FUNCTION_BLOCK FB_MachineControl EXTENDS FB_UniversalMachine IMPLEMENTS I_MachineControl
VAR PERSISTENT
	sLastLoadedRecipe						: STRING;
	sLastProductOrder						: STRING;
	(* Parameter have to adjust for Sorting Station *)
	lrSortGoodDistance			: LREAL := -24.0;	(* Distance between cam7 to sort station *)
	lrSortDirtDistance			: LREAL := -55.0;	(* Distance between cam7 to sort station *)
	lrSortDentDistance			: LREAL := -55.0;	(* Distance between cam7 to sort station *)
	lrSortRejectDistance		: LREAL := -60.0;	(* Distance between cam7 to sort station *)
	tSortValveGoodTime			: TIME := T#1000MS;		(* During time to shoot sample *)
	tSortValveDirtTime			: TIME := T#2000MS;		(* During time to shoot sample *)
	tSortValveDentTime			: TIME := T#1000MS;		(* During time to shoot sample *)
	tSortValveRejectTime		: TIME := T#1000MS;		(* During time to shoot sample *)
	
	rBowlFeederSetpoint 		: REAL := 60.0;
END_VAR
VAR	
	(* Process data *)
	//{attribute 'OPC.UA.DA' := '1	'}
	stBatchPerformance		: ST_BatchPerformacne; 	(* Data about performance about current proccesed batch *)
	//{attribute 'OPC.UA.DA' := '1	'}                                                          		
	stBatchData				: ST_BatchData;			(* Data about batch that is going to be processed*)

	(*--- Module Interface ---*)
	fbRobot 					: FB_Robot;
	fbRTCVision 				: FB_RTCVision;
	fbBowlFeeder				: FB_BowlFeeder;
	fbRotaryTable				: FB_AxisServo;
	
	(* Utilities *)
	fbPlcUps					: FB_UpsCx51xx;	
	
	(* IO PLC connect *)
	diProductPresenceBowl		: FB_DigitalInput;	(* *)
	diProductPresenceRobot		: FB_DigitalInput;	(* *)	
	
	poDoorLock					: FB_DigitalOutput;			(* Requests all machine lock's to close *)
	poResetButtonLight			: FB_DigitalOutput;			(* Physical reset button attached to door's of electrical cabinet *)
	
	doBlowBowlFeeder			: FB_DigitalOutput;
	doBlowGood					: FB_DigitalOutput;
	doBlowReject				: FB_DigitalOutput;
	doBlowDentContamination		: FB_DigitalOutput;
	doBlowDirtScratch			: FB_DigitalOutput;
	
	doTriggerCam1				: FB_DoubleTrigger;
	doTriggerCam2				: FB_DoubleTrigger;
	doTriggerCam3				: FB_DoubleTrigger;
	doTriggerCam4				: FB_DoubleTrigger;
	doTriggerCam5				: FB_DoubleTrigger;
	doTriggerCam6				: FB_DoubleTrigger;
	doTriggerCam7				: FB_DoubleTrigger;
	
	
	
	(* Auxilary *)
	tonDelay					: TON;				(* Provides any delay into the machine when switching something On/Off *)
	//tonTestDelay	: TON;	(* Delay which allows to see any page changes during tests *)	
	
	(* Parameter *)
	lrHOME_POSTION				: LREAL := 0.0;		(* Homming position *)
	stRotaryTableHomingOptions	: ST_HomingOptions;
	
	(* #ManualToAuto *)             	                                                            		
	//bManualToAutoRotate					: BOOL;																            	
	bStop								: BOOL;	
		
	// =============== State machine ============================================================
	eMachineStateUninitialized						: E_MachineCtrlStateUninitialized;
	eMachineStateInit								: E_MachineCtrlStateInit;
	eMachineStateAuto								: E_MachineCtrlStateAuto;
	eMachineStateAutoAOI							: E_MachineCtrlStateAutoAOI;
	eMachineStateAbort								: E_MachineCtrlStateAbort;
	eMachineStateManualToAuto						: E_MachineCtrlStateManualToAuto;
	
	(* HMI control *)
	btnStartBowl : BOOL;
	btnStopBowl : BOOL;
	
END_VAR

IF bFirstCycle THEN
	(* - bFirstCycle bit reset by parent *)
	(* --- Assign initial parameters for machine objects ---*)
	(* Assign UPS parameters *)
	fbPlcUps.MR_FirstCycle( 	sName 		:= 'PLC UPS',
								sNetID 		:= '',
								iPlcPort 	:= 851,
								tTimeout 	:= DEFAULT_ADS_TIMEOUT);
								
	(* Assign robots *)
	fbRobot.MR_FirstCycle(	sName				:= 'RH-3CRH4018-D-S15',
							iInitialOverride 	:= 3,					//low for testing
							sPLC_NET_ID 		:= '5.127.48.56.2.1',
							iCR800_1_ADDRESS 	:= 1020);
	
	(* Assign rotary table *)
	fbRotaryTable.MR_FirstCycle(	sName				:= sROTARY_TABLE_NAME,
									sMeasurementUnits	:= sROTARY_TABLE_MEASUREMENT_UNIT,
									bModulo				:= FALSE);
									
	fbRotaryTable.Override 			:= 100.0;
	fbRotaryTable.Velocity 			:= 100.0;	//400,325
	fbRotaryTable.Acceleration 		:= 1500.0; //1500,80|600
	fbRotaryTable.Deceleration 		:= 1500.0; //1500,800|600
	fbRotaryTable.Jerk 				:= 6000.0;//6000.0; //15000,8000|

	fbRotaryTable.JogPosition 		:= 0.0;
	fbRotaryTable.JogVelocity 		:= 300.0;
	fbRotaryTable.JogAcceleration 	:= 800.0;
	fbRotaryTable.JogDeceleration 	:= 800.0;
	fbRotaryTable.JogJerk 			:= 800.0;
	fbRotaryTable.StopDeceleration	:= 800.0;
	fbRotaryTable.StopJerk 			:= 8000.0;
	
	stRotaryTableHomingOptions.SearchDirection := Tc2_MC2.MC_Direction.MC_Negative_Direction;
	stRotaryTableHomingOptions.SearchVelocity 	:= 12.0;
	stRotaryTableHomingOptions.SyncDirection 	:= Tc2_MC2.MC_Direction.MC_Positive_Direction;
	stRotaryTableHomingOptions.SyncVelocity	:= 10.0;
	
	fbRotaryTable.HomingMode		:= MC_HomingMode.MC_DefaultHoming;
	fbRotaryTable.HomingOptions 	:= stRotaryTableHomingOptions;

	(* Assign bowl feeder *)
	fbBowlFeeder.MR_FirstCycle(sName := 'Bowl Feeder');
	fbBowlFeeder.Setpoint := 60.0;
	
	(* Assign RTC Vision system *)
	fbRTCVision.MR_FirstCycle(	sCameraName 	:= 'RTC Vision System',
								sClientHost		:= '10.20.254.8',
								sClientAmsNetID := '',
								iClientPort 	:= 23,
								tTimeout 		:= T#15S);
	
	(* Digital I/O *)
	diProductPresenceBowl.MR_FirstCycle(	sName := 'Product presence on bowl at pick point',
											sModuleType := '',
											sPortID := '');
											
	diProductPresenceRobot.MR_FirstCycle(	sName := 'Product presence at robot nozzle',
											sModuleType := '',
											sPortID := '');
									
	poDoorLock.MR_FirstCycle(		sName := 'Door lock station 1',
		                         sModuleType := '',
                                 sPortID := '');
								 
	poResetButtonLight.MR_FirstCycle(	sName := 'Reset Button light station 1',
										sModuleType := '',
										sPortID := '');

END_IF

(* Execute parent implementation *)
SUPER^();

(* --- Cyclic run ---*)
(* Cyclic run robots *)
fbRobot();
(* Cyclic run RTC vision *)
fbRTCVision();
(* Cyclic run bowl feeder *)
fbBowlFeeder();
(* Cyclic run rotary table *)
fbRotaryTable();
(* Utilities *)
fbPlcUps();

PROPERTY BowlFeeder : REFERENCE TO FB_BowlFeeder
GET
BowlFeeder REF= fbBowlFeeder;
END_GET
END_PROPERTY

METHOD PROTECTED GoldenSample : BOOL
VAR_INPUT
END_VAR
;
END_METHOD

METHOD PROTECTED M_AutoProcessing
VAR_INST
	(* Equipment module sequences *)
	BowlFeederProcess : UINT;
	RobotProcess : UINT;
	
	RotaryTableProcess : UINT;
	TableRegister		: UINT;
	
	(* Parameters *)
	bIsRobotAtRotaryTable : BOOL;
	OneStep : LREAL := 10.00;
END_VAR
/// ======================= Bowl feeder process ======================= {{{
CASE BowlFeederProcess OF
	0:
		IF fbBowlFeeder.MR_Start() THEN
			BowlFeederProcess := 10;
		END_IF
		
	10:
		;
		
END_CASE
///}}}
/// ======================= Robot process ======================= {{{
CASE RobotProcess OF
	0://IDLE go bowl
		fbRobot.MR_GoBowl();
		IF NOT fbRobot.Busy THEN
			RobotProcess := 5;
		END_IF
		
	5://Goto input
		IF diProductPresenceBowl.In THEN (* waiting product *)
			fbRobot.MR_GoInputProduct();
			IF NOT fbRobot.Busy THEN
				RobotProcess := 6;
			END_IF
		END_IF
	
	6://robot pick
		fbRobot.MR_Pick();
		IF NOT fbRobot.Busy THEN
			RobotProcess := 10;
		END_IF 
		
	10://go to station 1
		fbRobot.MR_GoStation1();
		IF NOT fbRobot.Busy THEN
			RobotProcess := 20;
		END_IF
	20:
		fbRTCVision.M_CommandStation1(DelayTimeForSecondTrigger := T#1MS);
		IF NOT fbRTCVision.Busy THEN
			RobotProcess := 30;
		END_IF
	30:
		fbRobot.MR_GoStation2();
		IF NOT fbRobot.Busy THEN
			RobotProcess := 40;
		END_IF
	40:
		fbRTCVision.M_CommandStation2(DelayTimeForSecondTrigger := T#34MS);
		IF NOT fbRTCVision.Busy THEN
			RobotProcess := 50;
		END_IF
	50:
		fbrobot.MR_GoRotaryTable();
		IF NOT fbrobot.Busy THEN
			RobotProcess:= 60;//waiting drop product
		END_IF
	
END_CASE

IF RobotProcess = 60 THEN
	bIsRobotAtRotaryTable := TRUE;
ELSE
	bIsRobotAtRotaryTable := FALSE;
END_IF

///}}}
///(*======================= Rotary Table process =======================*){{{
(* Product placed and reset robot sequence *)
CASE TableRegister OF
	0://take product from robot
		IF fbRotaryTable.Halted AND bIsRobotAtRotaryTable THEN
			fbrobot.MR_Place();
			IF NOT fbrobot.Busy THEN
				TableRegister := 10;
			END_IF
		END_IF
	10://buffer calc and add process
		IF Buffer_RotaryTable.Add2Data(in1 := fbRotaryTable.ActualPosition + OneStep, in2 := fbRotaryTable.ActualPosition + 2*OneStep) THEN
			IF Buffer_Station3.Add1Data(in := fbRotaryTable.ActualPosition + OneStep) THEN
				IF Buffer_Station4.Add1Data(in := fbRotaryTable.ActualPosition + 2*OneStep) THEN
					TableRegister := 20;

				END_IF				
			END_IF
		END_IF
END_CASE


(* Table sequences *)
CASE RotaryTableProcess OF
	0://Idle
		IF Buffer_RotaryTable.Count > 0 THEN
			RotaryTableProcess := 10;
		END_IF
	10:
		fbRotaryTable.MR_MoveRelative(lrRelativeDistance := Buffer_RotaryTable.GetValue);
		IF NOT fbRotaryTable.Busy THEN
//			iRTCVision.M_CommandStation1(); // change to station 3
//			IF NOT iRTCVision.Busy THEN
//				;
//			END_IF
			;
		END_IF
END_CASE
///}}}
END_METHOD

METHOD MR_Start : BOOL
(* 
Button START on the HMI
*)
fbMsgAutoStarted.Send(0);

IF eMachineStateAuto = MACHINE_STATE_AUTO_IDLE THEN
	eMachineState := MACHINE_STATE_AUTO;
	eMachineStateAuto := MACHINE_STATE_AUTO_RUNNING;
	bStop := FALSE;
	
END_IF

MR_Start := TRUE;
END_METHOD

METHOD MR_Stop : BOOL
VAR_INPUT
END_VAR
bRunning := FALSE;

IF eMachineStateAuto = MACHINE_STATE_AUTO_RUNNING THEN
	eMachineStateAuto := MACHINE_STATE_AUTO_IDLE;
	
END_IF
END_METHOD

METHOD PROTECTED MS_Aborting
(* 
Add here code to abort all machine objects's e.g robots, axes, cylinders. 
At the end add "eMachineState := MACHINE_STATE_UNINITIALIZED;" to finish aborting.
*)
CASE eMachineStateAbort OF
	MACHINE_STATE_ABORTING_TABLE:
		fbRotaryTable.MR_Abort();
		IF NOT fbRotaryTable.Active THEN
			eMachineState := MACHINE_STATE_UNINITIALIZED;
		eMachineStateUninitialized := MACHINE_STATE_UNINITIALIZED_DONE;
		END_IF
		
	MACHINE_STATE_ABORTING_ROBOT_CYCLE_STOP:
		IF fbRobot.ref_CR800.ErrorOccuring THEN			
			eMachineStateAbort := MACHINE_STATE_ABORTING_TABLE;
			eMachineState := MACHINE_STATE_UNINITIALIZED;
			eMachineStateUninitialized := MACHINE_STATE_UNINITIALIZED_DONE;
		ELSE
			fbRobot.ref_CR800.MR_CycleStop();
			IF NOT fbRobot.ref_CR800.Busy THEN
				eMachineStateAbort := MACHINE_STATE_ABORTING_TABLE;
				eMachineState := MACHINE_STATE_UNINITIALIZED;
				eMachineStateUninitialized := MACHINE_STATE_UNINITIALIZED_DONE;
			END_IF
		END_IF

END_CASE
END_METHOD

METHOD PROTECTED MS_Auto
VAR_INST
	bSetSP:BOOL;
	rSp:REAL;
END_VAR
CASE eMachineStateAuto OF
	MACHINE_STATE_AUTO_IDLE:
		bRunning := FALSE;
		
	MACHINE_STATE_AUTO_RUNNING:
		bRunning := TRUE;
		//Test();
		Production_fixing();
		//Robot_Process();
		//TableProcess();
		//tableRefer();
		//robotcamtest();
		//Robot_Process();
		
END_CASE

(*========== HMI control =============*)
(* Bowl feeder *)
IF btnStartBowl THEN
	fbBowlFeeder.MR_Start();
	doBlowBowlFeeder.Out := TRUE;
END_IF

IF btnStopBowl THEN
	fbBowlFeeder.MR_Stop();
	doBlowBowlFeeder.Out := FALSE;
END_IF

fbBowlFeeder.Setpoint := rBowlFeederSetpoint;
END_METHOD

METHOD PROTECTED MS_AutoToManual
VAR_INPUT
END_VAR
(* 
Add here code to switch machine into manual mode. 
At the end add "eMachineState := MACHINE_STATE_MANUAL;" to finish switching.
*)
(* Switching mode to manual simulation - DELETE *)
//tonTestDelay(IN := TRUE, PT:= T#500MS);
//bRunning := FALSE;
//IF tonTestDelay.Q THEN
//	tonTestDelay(IN := FALSE);
//	eMachineState := MACHINE_STATE_MANUAL;
//END_IF

bRunning := FALSE;
eMachineState := MACHINE_STATE_MANUAL;
END_METHOD

METHOD PROTECTED MS_Emergency
VAR_INPUT
END_VAR
END_METHOD

METHOD PROTECTED MS_Initializing
VAR_INST
	uBowlFeederInitState : UINT;
	uTableInitState : UINT;
	uVisionInitState : UINT;
	
END_VAR
(* 
Add here code to initialize all machine objects's e.g robots, axes, cylinders. 
At the end add "eMachineState := MACHINE_STATE_READY_INITIALIZED;" to finish initialization.
*)
CASE eMachineStateInit OF
	MACHINE_STATE_INITIALIZING_MACHINE_LOGGER:
		fbMachineLogger.MR_Init();
		IF NOT fbMachineLogger.Busy THEN
			eMachineStateInit := MACHINE_STATE_INITIALIZING_ROBOT_CONTROLERS_RESET;
		END_IF
(*	
	MACHINE_STATE_INITIALIZING_RECIPES_MANAGER:
		IF stShell.stPlatform.ref_fbRecipesManager.Active THEN
			eMachineStateInit := MACHINE_STATE_INITIALIZING_CLEAR_ALL_ERRORS;
		END_IF
		
	MACHINE_STATE_INITIALIZING_CLEAR_ALL_ERRORS:
		stShell.stPlatform.ref_fbAlarmControler.MR_ClearAll(TRUE);
		IF NOT stShell.stPlatform.ref_fbAlarmControler.Busy THEN
			//eMachineStateInit := MACHINE_STATE_INITIALIZING_MES_COMMAND_LOGGER;
			eMachineStateInit := MACHINE_STATE_INITIALIZING_SAFETY_INITIALIZATION;
		END_IF
	
	MACHINE_STATE_INITIALIZING_SAFETY_INITIALIZATION:
		stShell.stPlatform.ref_MachineSafety.RunStop := TRUE;
		tonDelay( IN := TRUE, PT := T#3S);
		IF tonDelay.Q THEN
			tonDelay(IN := FALSE);
			//fbMessageSafetySystemRestarted.Send(0); (* TC_Alarm *)
			eMachineStateInit := MACHINE_STATE_INITIALIZING_CHECK_ESTOP;
		END_IF
	
	MACHINE_STATE_INITIALIZING_CHECK_ESTOP:
		poDoorLock.Out := FALSE;
		IF stShell.stPlatform.ref_MachineSafety.E_Stop AND stShell.stPlatform.ref_MachineSafety.ExternalE_Stop THEN
			eMachineStateInit := MACHINE_STATE_INITIALIZING_CHECK_DOOR_LOCKS;
		END_IF
	
	MACHINE_STATE_INITIALIZING_CHECK_DOOR_LOCKS:
		IF NOT stShell.stPlatform.ref_MachineSafety.E_Stop OR NOT stShell.stPlatform.ref_MachineSafety.ExternalE_Stop THEN
			eMachineStateInit := MACHINE_STATE_INITIALIZING_CHECK_ESTOP;		
		ELSE
			IF stShell.stPlatform.ref_MachineSafety.SafetyOverride THEN
				eMachineStateInit := MACHINE_STATE_INITIALIZING_ROBOTS_POWER_CHECK;
			ELSE
				poDoorLock.Out := TRUE;
				IF stShell.stPlatform.ref_MachineSafety.DoorLock THEN
					eMachineStateInit := MACHINE_STATE_INITIALIZING_ROBOTS_POWER_CHECK;
				END_IF
			END_IF
		END_IF
	
	MACHINE_STATE_INITIALIZING_ROBOTS_POWER_CHECK:
		IF fbRobot.ref_CR800.CR800PoweredOn THEN
			eMachineStateInit := MACHINE_STATE_INITIALIZING_SAFETY_RESET;
		END_IF
	
	MACHINE_STATE_INITIALIZING_SAFETY_RESET:
		stShell.stPlatform.ref_MachineSafety.ErrorAck := TRUE;
		eMachineStateInit := MACHINE_STATE_INITIALIZING_SAFETY_START;
	
	MACHINE_STATE_INITIALIZING_SAFETY_START:
		stShell.stPlatform.ref_MachineSafety.ErrorAck := FALSE;
		IF NOT stShell.stPlatform.ref_MachineSafety.E_Stop OR NOT stShell.stPlatform.ref_MachineSafety.ExternalE_Stop THEN
			eMachineStateInit := MACHINE_STATE_INITIALIZING_CHECK_ESTOP;		
		ELSIF NOT stShell.stPlatform.ref_MachineSafety.SafetyOverride AND NOT stShell.stPlatform.ref_MachineSafety.DoorLock THEN
			eMachineStateInit := MACHINE_STATE_INITIALIZING_CHECK_DOOR_LOCKS;
		ELSE
			poResetButtonLight.Out := TRUE;
			IF stShell.stPlatform.ref_MachineSafety.RestartButton THEN
				poResetButtonLight.Out := FALSE;
				eMachineStateInit := MACHINE_STATE_INITIALIZING_ROBOT_CONTROLERS_RESET;
			END_IF
		END_IF
	*)
	MACHINE_STATE_INITIALIZING_ROBOT_CONTROLERS_RESET:
		fbRobot.ref_CR800.MR_Reset();
		IF NOT fbRobot.ref_CR800.Busy THEN
			uTableInitState := 10;
			uBowlFeederInitState := 10;
			eMachineStateInit := MACHINE_STATE_INITIALIZING_ROBOT_AUTO_MODE_SW;
		END_IF
(*
	MACHINE_STATE_INITIALIZING_SAFETY_CHECK:
		IF NOT stShell.stPlatform.ref_MachineSafety.FB_Error AND NOT stShell.stPlatform.ref_MachineSafety.FB_Error THEN
			fbRobot.ModeSwitch := TRUE;
			eMachineStateInit := MACHINE_STATE_INITIALIZING_ROBOT_ABORT;
		END_IF
	*)
	
	MACHINE_STATE_INITIALIZING_ROBOT_AUTO_MODE_SW:
		fbRobot.ModeSwitch := TRUE;
		eMachineStateInit := MACHINE_STATE_INITIALIZING_ROBOT_ABORT;
		
	MACHINE_STATE_INITIALIZING_ROBOT_ABORT:
		fbRobot.MR_Abort();
		IF NOT fbRobot.Active THEN
			eMachineStateInit := MACHINE_STATE_INITIALIZING_ROBOT_INIT;
		END_IF
	
	MACHINE_STATE_INITIALIZING_ROBOT_INIT:
		fbRobot.MR_Init();
		IF fbRobot.Active THEN
			eMachineStateInit := MACHINE_STATE_INITIALIZING_ROBOT_HOME;
		END_IF
	
	MACHINE_STATE_INITIALIZING_ROBOT_HOME:
		fbRobot.MR_GoHome();
		IF NOT fbRobot.Busy THEN
			eMachineStateInit := MACHINE_STATE_INITIALIZING_ROBOT_AUTOMATIC_MODE;
		END_IF
	
	MACHINE_STATE_INITIALIZING_ROBOT_AUTOMATIC_MODE:
		fbRobot.ref_CR800.MR_GoAuto();
		IF NOT fbRobot.ref_CR800.Busy THEN
			eMachineStateInit := MACHINE_STATE_INITIALIZING_DONE;
		END_IF
	
//	MACHINE_STATE_INITIALIZING_ROTARY_TABLE_ABORT:
		

//	MACHINE_STATE_INITIALIZING_ROTARY_TABLE_INIT:
		

//	MACHINE_STATE_INITIALIZING_ROTARY_TABLE_HOME:
		
		
//	MACHINE_STATE_INITIALIZING_BOWL_INIT:
		

	MACHINE_STATE_INITIALIZING_DONE:
		IF uTableInitState = 30 AND uBowlFeederInitState = 20 THEN	(* check Table and bowl init done *)
			eMachineStateInit := MACHINE_STATE_INITIALIZING_MACHINE_LOGGER;
			eMachineState := MACHINE_STATE_READY_INITIALIZED;
		END_IF
		
END_CASE
/////////////////////////////////////////////////////////
CASE uTableInitState OF
	0://idle
		;
	5:
		fbRotaryTable.MR_Abort();
		IF NOT fbRotaryTable.PowerOn THEN
			uTableInitState := 10;
		END_IF
	10://init
		fbRotaryTable.MR_Init();
		IF fbRotaryTable.PowerOn THEN
			uTableInitState := 20;
		END_IF
	20://homing
		fbRotaryTable.MR_Home(lrHomePosition := DEFAULT_HOME_POSITION );
		IF fbRotaryTable.IsHomed THEN
			uTableInitState := 30;
		END_IF
	30://done
		;
END_CASE
/////////////////////////////////////////////////////////
CASE uBowlFeederInitState OF
	0://idle
		;
	10:
		fbBowlFeeder.MR_Init();
		IF NOT fbBowlFeeder.Busy THEN
			uBowlFeederInitState := 20;
		END_IF
	20://done
		;
END_CASE
END_METHOD

METHOD PROTECTED MS_Manual
VAR_INPUT
END_VAR
(* 
Leave empty - manual mode is provided by HMI controler and automatic frame generator.
*)
;
END_METHOD

METHOD PROTECTED MS_ManualToAuto
VAR_INPUT
END_VAR
(* 
Add here code to switch machine into auto mode. 
At the end add "eMachineState := MACHINE_STATE_AUTO;" to finish switching.
*)
//CASE eMachineStateManualToAuto OF
//	MACHINE_STATE_MANUAL_TO_AUTO_ROBOT_CYCLE_STOP:
//		IF arrRobot[0].ErrorOccuring THEN
//			eMachineStateManualToAuto := MACHINE_STATE_MANUAL_TO_AUTO_ROBOT_ABORT;
//		ELSE
//			arrRobot[0].MR_CycleStop();
//			IF NOT arrRobot[0].Busy THEN
//				eMachineStateManualToAuto := MACHINE_STATE_MANUAL_TO_AUTO_ROBOT_ABORT;
//			END_IF
//		END_IF
		
//	MACHINE_STATE_MANUAL_TO_AUTO_ROBOT_ABORT:
//		arrRobot[0].MR_Abort();
//		IF NOT arrRobot[0].Active THEN
//			//eMachineStateManualToAuto := MACHINE_STATE_MANUAL_TO_AUTO_ROBOT_REMOTE_MODE;
//			eMachineStateManualToAuto := MACHINE_STATE_MANUAL_TO_AUTO_ROBOT_INIT;
//		END_IF
	
////	MACHINE_STATE_MANUAL_TO_AUTO_ROBOT_REMOTE_MODE:
////		poRobotModeSwitch.Out := TRUE;
////		tonDelay( IN := TRUE, PT:= T#500MS);
////		IF tonDelay.Q THEN
////			tonDelay(IN := FALSE);
////			eMachineStateManualToAuto := MACHINE_STATE_MANUAL_TO_AUTO_ROBOT_ONE_INIT;
////		END_IF
		
//	MACHINE_STATE_MANUAL_TO_AUTO_ROBOT_INIT:
//		arrRobot[0].MR_Init();
//		IF arrRobot[0].Active THEN
//			eMachineStateManualToAuto := MACHINE_STATE_MANUAL_TO_AUTO_ROBOT_HOME;
//		END_IF
		
//	MACHINE_STATE_MANUAL_TO_AUTO_ROBOT_HOME:
//		arrRobot[0].MR_GoHome();
//		IF NOT arrRobot[0].Busy THEN
//			eMachineStateManualToAuto := MACHINE_STATE_MANUAL_TO_AUTO_ROBOT_AUTOMATIC_MODE;
//		END_IF
		
//	MACHINE_STATE_MANUAL_TO_AUTO_ROBOT_AUTOMATIC_MODE:
//		arrRobot[0].MR_GoAuto();
//		IF NOT arrRobot[0].Busy THEN
//			eMachineStateManualToAuto := MACHINE_STATE_MANUAL_TO_AUTO_DONE;
//		END_IF
		
//	MACHINE_STATE_MANUAL_TO_AUTO_DONE:
//		eMachineStateManualToAuto := MACHINE_STATE_MANUAL_TO_AUTO_ROBOT_CYCLE_STOP;
//		eMachineState := MACHINE_STATE_AUTO;
		
//END_CASE
END_METHOD

METHOD PROTECTED MS_ReadyInitialized
VAR_INPUT
END_VAR
(*
Add code here if some internal parameters are needed to set after initialization or leave it default.
At the end add "eMachineState := MACHINE_STATE_AUTO;" to finish and go to IDLE state.
*)
eMachineStateInit := MACHINE_STATE_INITIALIZING_MACHINE_LOGGER;
eMachineState := MACHINE_STATE_AUTO;
eMachineStateAuto := MACHINE_STATE_AUTO_IDLE;
eMachineStateAutoAOI := MACHINE_STATE_AUTO_AOI_IDLE;
END_METHOD

METHOD PROTECTED MS_Reset
VAR_INPUT
END_VAR
(* 
Add here code to reset all machine objects's e.g robots, axes, cylinders. 
At the end add "eMachineState := MACHINE_STATE_RESET_DONE;" to finish reseting.
*)
(* Reset simulation - DELETE  *)
//tonTestDelay(IN := TRUE, PT:= T#4S);
//IF tonTestDelay.Q THEN
//	tonTestDelay(IN := FALSE);
//	eMachineState := MACHINE_STATE_RESET_DONE;
//END_IF

eMachineState := MACHINE_STATE_RESET_DONE;
END_METHOD

METHOD PROTECTED MS_ResetDone
VAR_INPUT
END_VAR
eMachineState := eMachineStateBeforeReset;
END_METHOD

METHOD PROTECTED MS_Uninitialized

VAR_INST
	btestmethodcam: BOOL;
	btestasd : bool;
END_VAR
VAR
	
END_VAR
CASE eMachineStateUninitialized OF
	
	MACHINE_STATE_UNINITIALIZED_POWER_ON_CR800:
		IF fbRobot.ref_CR800.CR800PoweredOn THEN
			eMachineStateUninitialized := MACHINE_STATE_UNINITIALIZED_CR800_ETHERCAT_STATUS_CHECK;
		END_IF
	
	MACHINE_STATE_UNINITIALIZED_CR800_ETHERCAT_STATUS_CHECK:
		IF fbRobot.M_EtherCATStatusCheck() THEN
			eMachineStateUninitialized := MACHINE_STATE_UNINITIALIZED_DONE;
		END_IF

	MACHINE_STATE_UNINITIALIZED_DONE:
		eMachineStateInit := MACHINE_STATE_INITIALIZING_MACHINE_LOGGER;
	
END_CASE
END_METHOD

METHOD PROTECTED Production : BOOL
VAR_INST
	(* Robot *)
	RobotState 					: UINT;
	
	(* Table *)
	TableState					: UINT;
	OneStep 					: LREAL:= -60.0; //-61.1928;	(* Define by the distance between station 3 and 4 *)
	lrRelativeDistance 			: LREAL;
	bProductAboveTable 			: BOOL;				(* Signal Robot is at the table *)
	bGetPictureStation3			: BOOL; 			(* Cmd get picture st3 to vision system *)
	bGetPictureStation4 		: BOOL; 			(* Cmd get picture st4 to vision system *)
	bResultProcessing 			: BOOL;				(* Request result from vision system, then add buffer for sorting station *)
	
	(* Buffer *)
	BufferState : UINT;
	Buffer_RotaryTable			: FB_DataSetFifo_1; 	(* Contain the position of all product on the table *)
	Buffer_Station3				: FB_DataSetFifo_1;	(* Contain the trigger position *)
	Buffer_Station4				: FB_DataSetFifo_1;	(* Contain the trigger position *)
	
	(* Sorting Station *)
	Buffer_SortGood				: FB_DataSetFifo_1;
	Buffer_SortDirt				: FB_DataSetFifo_1;
	Buffer_SortDent				: FB_DataSetFifo_1;
	Buffer_SortReject			: FB_DataSetFifo_1;
	
	
	
	lrSortGoodPos				: LREAL;
	lrSortDirtPos				: LREAL;
	lrSortDentPos				: LREAL;
	lrSortRejectPos				: LREAL;
	
	uSortGoodGetPosState		: UINT; 			(* state machine of get sort position from buffer *)
	uSortDirtGetPosState		: UINT;
	uSortDentGetPosState		: UINT;
	uSortRejectGetPosState		: UINT;
		
	tonGoodDelay				: TON;				(* one shoot of good delay valve *)
	tonDirtDelay				: TON;				(* one shoot of dirt delay valve *)
	tonDentDelay				: TON;				(* one shoot of dent delay valve *)								
	tonRejectDelay				: TON;				(* one shoot of reject delay valve *)	
							

	
	(*=== Vision ===*)
	Vision3State 		: UINT;
	Vision4State		: UINT;
	lrCapPosStation3 	: LREAL;
	lrCapPosStation4	: LREAL;
	bGood 				: BOOL;
	bAtVision3 			: BOOL;	(* Product is at vision 3 *)
	bAtVision4 			: BOOL;	(* Product is at vision 4 *)
	eFinalResult		: E_VisionResult;

	(* Axis status flags *)
	bActive					: BOOL;
	bBusy					: BOOL;								(* Function block currently executes one of the requests *)
	bError					: BOOL;								(* Error status flag *)
	iErrorID				: UDINT;							(* Error ID *)
	iAxisErrorID			: UDINT;							(* Axis error ID*)
	lrActualPosition		: LREAL;							(* Actual axis position in selected units *)
	rActualVelocity			: REAL;								(* Actual axis velocity in selected units *)
	bPowerOn 				: BOOL;								(* Power On status bit *)
	bIsHomed				: BOOL;								(* Axis has been homed even once *)
	bInVelocity				: BOOL;								(* Axis is moving in target velocity *)
	bInPostion				: BOOL;								(* Axis reached target position *)
	bMoveActive				: BOOL;								(* Axis is moving to target position *)
	bJogDone				: BOOL;								(* Axis manual movement by jog done *)
	bStopped				: BOOL;								(* Axis movement has been stopped *)
	bHalted					: BOOL;								(* Axis movement has been halted *)
	eStatePlcOpen			: E_AxisStatePlcOpen;
	
	uBufferTableCount : UDINT;
	
	(* testing bit *)
	bResultTest : BOOL;
	bResultGood : BOOL;
	bResultDirt : BOOL;
	bResultDent : BOOL;
	bResultReject : BOOL;

END_VAR
///(*==================================== Robot + Vision process ====================================*){{{
CASE RobotState OF	
	0://IDLE go bowl
		fbRobot.MR_GoBowl();
		IF NOT fbRobot.Busy THEN
			RobotState := 5;
		END_IF		
	5://product detected
		IF diProductPresenceBowl.In THEN (* waiting product *)
			RobotState := 6;
		END_IF
	
	6://go input
		fbRobot.MR_GoInputProduct();
		IF NOT fbRobot.Busy THEN
			RobotState := 7;
		END_IF
		
	7://robot pick
		fbRobot.MR_Pick();
		IF NOT fbRobot.Busy THEN
			RobotState := 10;
		END_IF 
		
	10://go to station 1
		fbRobot.MR_GoStation1();
		IF NOT fbRobot.Busy THEN
			RobotState := 20;
		END_IF
		
	20://double trig cam 1+2
		IF doTriggerCam1.Command(PulseWidth:=T#1MS, DelayTimeForSecondTrigger := T#35MS) AND
			doTriggerCam2.Command(PulseWidth:=T#1MS, DelayTimeForSecondTrigger := T#35MS) THEN
			RobotState:= 30;
		END_IF
	30://go to station 2
		fbRobot.MR_GoStation2();
		IF NOT fbRobot.Busy THEN
			RobotState := 40;
		END_IF
	40://double trig cam 3+4
		IF doTriggerCam3.Command(PulseWidth:=T#1MS, DelayTimeForSecondTrigger := T#35MS) AND
			doTriggerCam4.Command(PulseWidth:=T#1MS, DelayTimeForSecondTrigger := T#35MS) THEN
			RobotState := 50;
		END_IF
	50://goto rotary table
		fbRobot.MR_GoRotaryTable();
		IF NOT fbRobot.Busy THEN
			bProductAboveTable := TRUE;		
			RobotState:= 60;
		END_IF
	60://waiting command from table
		;
		
END_CASE
///============================================================================================}}}
///(*==================================== Table process ====================================*){{{
CASE TableState OF
	0:// idle | waiting for product
		IF bProductAboveTable THEN
			TableState:= 10;
		END_IF
	10://command place product and reset robot sequence
		fbRobot.MR_Place();
		IF NOT fbRobot.Busy THEN
			bProductAboveTable := FALSE;
			RobotState := 0;
			TableState := 20;
		END_IF
	20://add buffer for st 3+4, table
		Buffer_RotaryTable.A_Add(in:= OneStep);
		Buffer_RotaryTable.A_Add(in:= OneStep);
		Buffer_Station3.A_Add(in:= fbRotaryTable.ActualPosition + OneStep);
		Buffer_Station4.A_Add(in:= fbRotaryTable.ActualPosition + 2*OneStep);
		TableState := 30;
		
//	21://get vision 3capture position
//		IF Vision3State = 0 THEN
//			Vision3State:= 10;
//			TableState:=22;
//		END_IF
//	22://get vision 4 capture position
//		IF Vision4State = 0 THEN
//			Vision4State:= 10;
//			TableState:=30;
//		END_IF
	
	30://get table distance movement
		Buffer_RotaryTable.A_Remove(out => lrRelativeDistance);
		TableState := 40;
	40://move distance
		fbRotaryTable.MR_MoveRelative(lrRelativeDistance);
		IF fbRotaryTable.InPosition THEN
			
			TableState := 41;
		END_IF
		
	41:// check position of vision station 3
		IF Vision3State = 0 THEN
			TableState := 42;
		END_IF
	42:
		Buffer_Station3.A_Get(out => lrCapPosStation3);
		bGetPictureStation3 := TRUE;
		
		IF LREAL_TO_INT(fbRotaryTable.ActualPosition) = LREAL_TO_INT(lrCapPosStation3) THEN
			Buffer_Station3.A_Remove(out => lrCapPosStation3);
			Vision3State:= 30;
			TableState := 43;
			
		ELSE
			bGetPictureStation3 := FALSE;
			TableState := 43;
			
		END_IF
			
	43:// check position of vision station 4
		IF Vision4State = 0 THEN
			TableState := 44;
		END_IF
	44:
		Buffer_Station4.A_Get(out => lrCapPosStation4);
		bGetPictureStation4 := TRUE;
		bResultProcessing := TRUE;
		
		IF LREAL_TO_INT(fbRotaryTable.ActualPosition) = LREAL_TO_INT(lrCapPosStation4) THEN
			Buffer_Station4.A_Remove(out => lrCapPosStation4);
			Vision4State:= 30;
			TableState := 60;
			
		ELSE
			bGetPictureStation4 := FALSE;
			bResultProcessing := FALSE;
			TableState := 60;
			
		END_IF
	
	
	
	
//	50://command vision 3
//		IF Vision3State = 0 THEN
//			Vision3State:= 20;
//			TableState:=55;
//		END_IF
//	55:	//command vision 4
//		IF Vision4State = 0 THEN
//			Vision4State:= 20;
//			TableState:=60;
//		END_IF

	
	
	
	
	60://check taking picture done
		IF NOT bGetPictureStation3 AND NOT bGetPictureStation4  AND NOT bResultProcessing THEN
			TableState := 70;
		END_IF
		
	70://state check result | product above table | buffer | go through sorting station
		IF bProductAboveTable THEN
			TableState := 10;//take product
		ELSIF Buffer_RotaryTable.nCount > 0 THEN
			TableState := 30;//get distance
		ELSE
			(* Make sure that the product is sorted *)
			fbRotaryTable.MR_MoveRelative(2*OneStep);
			IF fbRotaryTable.InPosition THEN
				
				TableState := 0;
			END_IF
			
		END_IF
	
END_CASE
///============================================================================================}}}
///(*==================================== Vision 3+4 process ====================================*){{{
CASE Vision3State OF
	0://idle | waiting
		;
//	10://get position in buffer
//		Buffer_Station3.A_Remove(out => lrCapPosStation3);
//		Vision3State := 0;

//	20://check position with table
//		bGetPictureStation3 := TRUE;
//		IF LREAL_TO_INT(fbRotaryTable.ActualPosition) = LREAL_TO_INT(lrCapPosStation3) THEN //convert from lreal to int for less precise
//			Vision3State:= 30;
//		ELSE
//			bGetPictureStation3 := FALSE;
//			Vision3State:= 0;
//		END_IF
			
	30://take picture cam 5+6
		IF doTriggerCam5.Command(PulseWidth:= T#1MS, DelayTimeForSecondTrigger:= T#34MS) AND
			doTriggerCam6.Command(PulseWidth:= T#1MS, DelayTimeForSecondTrigger:= T#34MS) THEN
			
			bGetPictureStation3 := FALSE;
			Vision3State := 0; 
		END_IF
		
END_CASE

(* station 4 have to take picture and request result from system *)
CASE Vision4State OF
	0:
		;
//	10://get trigger position in buffer
//		Buffer_Station4.A_Remove(out => lrCapPosStation4);
//		Vision4State := 0;

//	20://check trigger position with table position
//		bGetPictureStation4 := TRUE;
//		bResultProcessing 	:= TRUE;
//		IF LREAL_TO_INT(fbRotaryTable.ActualPosition) = LREAL_TO_INT(lrCapPosStation4) THEN //convert from lreal to int for less precise
//			Vision4State:= 30;
//		ELSE
//			bResultProcessing			:= FALSE;
//			bGetPictureStation4 		:= FALSE;
//			Vision4State:= 0;
//		END_IF
	
	30://trigger cam 7
		IF doTriggerCam7.Command(PulseWidth:= T#1MS, DelayTimeForSecondTrigger:= T#33MS) THEN
			bGetPictureStation4 := FALSE;
			Vision4State:= 40;
		END_IF
		
	40://request result
		(* testing purpose *)
		bResultGood:= TRUE;
		IF bResultGood THEN
			eFinalResult := VISION_RESULT_GOOD;
			bResultGood := FALSE;
			Vision4State:= 0;
		ELSIF bResultDirt THEN
			eFinalResult := VISION_RESULT_CONTAMINATION_DIRTY;
			bResultDirt := FALSE;
			Vision4State:= 0;
		ELSIF bResultDent THEN
			eFinalResult := VISION_RESULT_SCRATCH_DENT;
			bResultDent := FALSE;
			Vision4State:= 0;
		ELSIF bResultReject THEN
			eFinalResult := VISION_RESULT_REJECT;
			bResultReject := FALSE;
			Vision4State:= 0;
		END_IF

END_CASE
///============================================================================================}}}
///(*==================================== Sorting station ====================================*){{{
(* Add buffer for sorting station *)
CASE eFinalResult OF
	VISION_RESULT_UNKNOWN:
		;
	VISION_RESULT_GOOD:
		Buffer_SortGood.A_Add(in := fbRotaryTable.ActualPosition + lrSortGoodDistance);
		eFinalResult 		:= VISION_RESULT_UNKNOWN;
	VISION_RESULT_CONTAMINATION_DIRTY:
		Buffer_SortDirt.A_Add(in := fbRotaryTable.ActualPosition + lrSortDirtDistance);
		eFinalResult 		:= VISION_RESULT_UNKNOWN;
	VISION_RESULT_SCRATCH_DENT:
		Buffer_SortDent.A_Add(in := fbRotaryTable.ActualPosition + lrSortDentDistance);
		eFinalResult 		:= VISION_RESULT_UNKNOWN;
	VISION_RESULT_REJECT:
		Buffer_SortReject.A_Add(in := fbRotaryTable.ActualPosition + lrSortRejectDistance);
		eFinalResult 		:= VISION_RESULT_UNKNOWN;

END_CASE
(* Shoot the product out *)
(* Good case *)
CASE uSortGoodGetPosState OF
	0://idle | check buffer
		IF Buffer_SortGood.nCount > 0 THEN
			uSortGoodGetPosState:= 10;
		END_IF
	10://get position
		Buffer_SortGood.A_Get(out => lrSortGoodPos);
		uSortGoodGetPosState := 20;
	20://waiting table move in position | command table
		bResultProcessing 	:= FALSE;
		IF LREAL_TO_INT(fbRotaryTable.ActualPosition) <= LREAL_TO_INT(lrSortGoodPos) THEN
			uSortGoodGetPosState := 30;
		END_IF
	30://shoot it
		Buffer_SortGood.A_Remove(out => lrSortGoodPos);
		doBlowGood.Out := TRUE;
		uSortGoodGetPosState := 40;
		
	40://off
		tonGoodDelay(IN := TRUE, PT := tSortValveGoodTime);
		IF tonGoodDelay.Q THEN	
			doBlowGood.Out := FALSE;
			tonGoodDelay.IN := FALSE;
			uSortGoodGetPosState := 0;
		END_IF
		
END_CASE
(* DIRT CASE *)
CASE uSortDirtGetPosState OF
	0://idle | check buffer
		IF Buffer_SortDirt.nCount > 0 THEN
			uSortDirtGetPosState:= 10;
		END_IF
	10://get position
		Buffer_SortDirt.A_Get(out => lrSortDirtPos);
		uSortDirtGetPosState := 20;
	20://waiting table move in position | command table
		bResultProcessing 	:= FALSE;
		IF LREAL_TO_INT(fbRotaryTable.ActualPosition) <= LREAL_TO_INT(lrSortDirtPos) THEN
			uSortDirtGetPosState := 30;
		END_IF
	30://shoot it
		Buffer_SortDirt.A_Remove(out => lrSortDirtPos);
		doBlowDirtScratch.Out := TRUE;
		uSortDirtGetPosState := 40;
		
	40://off
		tonDirtDelay(IN := TRUE, PT := tSortValveDirtTime);
		IF tonDirtDelay.Q THEN	
			doBlowDirtScratch.Out := FALSE;
			tonDirtDelay.IN := FALSE;
			uSortDirtGetPosState := 0;
		END_IF
		
END_CASE
(* DENT CASE *)
CASE uSortDentGetPosState OF
	0://idle | check buffer
		IF Buffer_SortDent.nCount > 0 THEN
			uSortDentGetPosState:= 10;
		END_IF
	10://get position
		Buffer_SortDent.A_Get(out => lrSortDentPos);
		uSortDentGetPosState := 20;
	20://waiting table move in position | command table
		bResultProcessing 	:= FALSE;
		IF LREAL_TO_INT(fbRotaryTable.ActualPosition) <= LREAL_TO_INT(lrSortDentPos) THEN
			uSortDentGetPosState := 30;
		END_IF
	30://shoot it
		Buffer_SortDent.A_Remove(out => lrSortDentPos);
		doBlowDentContamination.Out := TRUE;
		uSortDentGetPosState := 40;
		
	40://off
		tonDentDelay(IN := TRUE, PT := tSortValveDentTime);
		IF tonDentDelay.Q THEN	
			doBlowDentContamination.Out := FALSE;
			tonDentDelay.IN := FALSE;
			uSortDentGetPosState := 0;
		END_IF
		
END_CASE
(* REJECT CASE *)
CASE uSortRejectGetPosState OF
	0://idle | check buffer
		IF Buffer_SortReject.nCount > 0 THEN
			uSortRejectGetPosState:= 10;
		END_IF
	10://get position
		Buffer_SortReject.A_Get(out => lrSortRejectPos);
		uSortRejectGetPosState := 20;
	20://waiting table move in position | command table
		bResultProcessing 	:= FALSE;
		IF LREAL_TO_INT(fbRotaryTable.ActualPosition) <= LREAL_TO_INT(lrSortRejectPos) THEN
			uSortRejectGetPosState := 30;
		END_IF
	30://shoot it
		Buffer_SortReject.A_Remove(out => lrSortRejectPos);
		doBlowReject.Out := TRUE;
		uSortRejectGetPosState := 40;
		
	40://off
		tonRejectDelay(IN := TRUE, PT := tSortValveRejectTime);
		IF tonRejectDelay.Q THEN	
			doBlowReject.Out := FALSE;
			tonRejectDelay.IN := FALSE;
			uSortRejectGetPosState := 0;
		END_IF
		
END_CASE
///============================================================================================}}}
(* control param *)
fbRobot.ref_CR800.Override:= 5;
uBufferTableCount:= Buffer_RotaryTable.nCount;

(* Mornitoring param *)
bActive 			:= fbRotaryTable.Active;
bBusy				:= fbRotaryTable.Busy;
bError 				:= fbRotaryTable.Error;
iErrorID 			:= fbRotaryTable.ErrorID;
iAxisErrorID 		:= fbRotaryTable.ErrorID;
lrActualPosition 	:= fbRotaryTable.ActualPosition;
rActualVelocity		:= fbRotaryTable.ActualVelocity;
bPowerOn 			:= fbRotaryTable.PowerOn;
bIsHomed 			:= fbRotaryTable.IsHomed;
bInVelocity			:= fbRotaryTable.InVelocity;
bInPostion 			:= fbRotaryTable.InPosition;
bMoveActive 		:= fbRotaryTable.MoveActive;
bJogDone 			:= fbRotaryTable.JogDone;
bStopped 			:= fbRotaryTable.Stopped;
bHalted 			:= fbRotaryTable.Halted;
eStatePlcOpen		:= fbRotaryTable.StatePlcOpen;

fbRobot.ref_CR800.Override:= 30;
fbRotaryTable.Velocity 			:= 50.0;
END_METHOD

METHOD PROTECTED Production_fixing : BOOL
VAR_INST
	(* Robot *)
	RobotState 					: UINT;
	
	(* Table *)
	TableState					: UINT;
	OneStep 					: LREAL:= -30.0; //-61.1928;	(* Define by the distance between station 3 and 4 *)
	lrRelativeDistance 			: LREAL;
	bProductAboveTable 			: BOOL;				(* Signal Robot is at the table *)
	bGetPictureStation3			: BOOL; 			(* Cmd get picture st3 to vision system *)
	bGetPictureStation4 		: BOOL; 			(* Cmd get picture st4 to vision system *)
	bResultProcessing 			: BOOL;				(* Request result from vision system, then add buffer for sorting station *)
	
	(* Buffer *)
	BufferState : UINT;
	Buffer_RotaryTable			: FB_DataSetFifo_1; 	(* Contain the position of all product on the table *)
	Buffer_Station3				: FB_DataSetFifo_1;	(* Contain the trigger position *)
	Buffer_Station4				: FB_DataSetFifo_1;	(* Contain the trigger position *)
	
	(* Sorting Station *)
	Buffer_SortGood				: FB_DataSetFifo_1;
	Buffer_SortDirt				: FB_DataSetFifo_1;
	Buffer_SortDent				: FB_DataSetFifo_1;
	Buffer_SortReject			: FB_DataSetFifo_1;
	
	
	
	lrSortGoodPos				: LREAL;
	lrSortDirtPos				: LREAL;
	lrSortDentPos				: LREAL;
	lrSortRejectPos				: LREAL;
	
	uSortGoodGetPosState		: UINT; 			(* state machine of get sort position from buffer *)
	uSortDirtGetPosState		: UINT;
	uSortDentGetPosState		: UINT;
	uSortRejectGetPosState		: UINT;
		
	tonGoodDelay				: TON;				(* one shoot of good delay valve *)
	tonDirtDelay				: TON;				(* one shoot of dirt delay valve *)
	tonDentDelay				: TON;				(* one shoot of dent delay valve *)								
	tonRejectDelay				: TON;				(* one shoot of reject delay valve *)	
							

	
	(*=== Vision ===*)
	Vision3State 		: UINT;
	Vision4State		: UINT;
	lrCapPosStation3 	: LREAL;
	lrCapPosStation4	: LREAL;
	bGood 				: BOOL;
	bAtVision3 			: BOOL;	(* Product is at vision 3 *)
	bAtVision4 			: BOOL;	(* Product is at vision 4 *)
	eFinalResult		: E_VisionResult;

	(* Axis status flags *)
	bActive					: BOOL;
	bBusy					: BOOL;								(* Function block currently executes one of the requests *)
	bError					: BOOL;								(* Error status flag *)
	iErrorID				: UDINT;							(* Error ID *)
	iAxisErrorID			: UDINT;							(* Axis error ID*)
	lrActualPosition		: LREAL;							(* Actual axis position in selected units *)
	rActualVelocity			: REAL;								(* Actual axis velocity in selected units *)
	bPowerOn 				: BOOL;								(* Power On status bit *)
	bIsHomed				: BOOL;								(* Axis has been homed even once *)
	bInVelocity				: BOOL;								(* Axis is moving in target velocity *)
	bInPostion				: BOOL;								(* Axis reached target position *)
	bMoveActive				: BOOL;								(* Axis is moving to target position *)
	bJogDone				: BOOL;								(* Axis manual movement by jog done *)
	bStopped				: BOOL;								(* Axis movement has been stopped *)
	bHalted					: BOOL;								(* Axis movement has been halted *)
	eStatePlcOpen			: E_AxisStatePlcOpen;
	
	uBufferTableCount : UDINT;
	
	(* testing bit *)
	bResultTest : BOOL;
	bResultGood : BOOL;
	bResultDirt : BOOL;
	bResultDent : BOOL;
	bResultReject : BOOL;

	(**)
	iTableSupervisor 	: UINT;
	iTableExecutor 		: UINT;
	
	Buffer_Sorting		: FB_DataSetFifo_1;	(* Contain the trigger position *)
	
	lrStation3Location : LREAL;
	lrStation4Location : LREAL;
	lrStationSortLocation : LREAL;
	lrTargetLocation : LREAL;
	
	bBufferTest : BOOL;
	
END_VAR
///(*==================================== Robot + Vision process ====================================*){{{
CASE RobotState OF	
	0://IDLE go bowl
		fbRobot.MR_GoBowl();
		IF NOT fbRobot.Busy THEN
			RobotState := 5;
		END_IF		
	5://product detected
		IF diProductPresenceBowl.In THEN (* waiting product *)
			RobotState := 6;
		END_IF
	
	6://go input
		fbRobot.MR_GoInputProduct();
		IF NOT fbRobot.Busy THEN
			RobotState := 7;
		END_IF
		
	7://robot pick
		fbRobot.MR_Pick();
		IF NOT fbRobot.Busy THEN
			RobotState := 10;
		END_IF 
		
	10://go to station 1
		fbRobot.MR_GoStation1();
		IF NOT fbRobot.Busy THEN
			RobotState := 20;
		END_IF
		
	20://double trig cam 1+2
		IF doTriggerCam1.Command(PulseWidth:=T#1MS, DelayTimeForSecondTrigger := T#35MS) AND
			doTriggerCam2.Command(PulseWidth:=T#1MS, DelayTimeForSecondTrigger := T#35MS) THEN
			RobotState:= 30;
		END_IF
	30://go to station 2
		fbRobot.MR_GoStation2();
		IF NOT fbRobot.Busy THEN
			RobotState := 40;
		END_IF
	40://double trig cam 3+4
		IF doTriggerCam3.Command(PulseWidth:=T#1MS, DelayTimeForSecondTrigger := T#35MS) AND
			doTriggerCam4.Command(PulseWidth:=T#1MS, DelayTimeForSecondTrigger := T#35MS) THEN
			RobotState := 50;
		END_IF
	50://goto rotary table
		fbRobot.MR_GoRotaryTable();
		IF NOT fbRobot.Busy THEN
			bProductAboveTable := TRUE;		
			RobotState:= 60;
		END_IF
	60://waiting command from table
		;
		
END_CASE
///============================================================================================}}}
(* TABLE SUPERVISOR *)
CASE iTableSupervisor OF
	0:
		IF bProductAboveTable THEN			
			IF iTableExecutor = 0 THEN//IDLE
				RobotState:=60;
			END_IF
		END_IF
		
END_CASE
(* TABLE EXECUTOR *)
CASE iTableExecutor OF
	0: //IDLE
		;
	10://TAKE PRODUCT
		
	20://ADD BUFFER
		Buffer_Station3.A_Add(in:= fbRotaryTable.ActualPosition + 2*OneStep); 	(* station position *)
		Buffer_Station4.A_Add(in:= fbRotaryTable.ActualPosition + 4*OneStep);	(* station position *)
		
		Buffer_RotaryTable.A_Add(in:= fbRotaryTable.ActualPosition + OneStep);	(* place position *)
		Buffer_RotaryTable.A_Add(in:= fbRotaryTable.ActualPosition + OneStep);	(* place position *)
		Buffer_RotaryTable.A_Add(in:= fbRotaryTable.ActualPosition + OneStep);	(* place position *)
		Buffer_RotaryTable.A_Add(in:= fbRotaryTable.ActualPosition + OneStep);	(* place position *)
		
		iTableExecutor := 30;
	30://calc the position
		IF Buffer_Station3.nCount > 0 AND Buffer_Station4.nCount > 0 THEN
			Buffer_Station3.A_Get(out => lrStation3Location);
			Buffer_Station4.A_Get(out => lrStation4Location);
			
			IF LREAL_TO_LINT(lrStation3Location) > LREAL_TO_LINT(lrStation4Location) THEN
				lrTargetLocation := lrStation3Location;
				Buffer_Station3.A_Remove(out => lrStation3Location);
				
			ELSIF LREAL_TO_LINT(lrStation3Location) < LREAL_TO_LINT(lrStation4Location) THEN
				lrTargetLocation := lrStation4Location;
				Buffer_Station4.A_Remove(out => lrStation4Location);
				
			ELSE
				lrTargetLocation := lrStation3Location;
				Buffer_Station3.A_Remove(out => lrStation3Location);
				Buffer_Station4.A_Remove(out => lrStation4Location);
			
			END_IF
			iTableExecutor := 40;
			
		ELSIF Buffer_Station3.nCount = 0 AND Buffer_Station4.nCount = 0 THEN
			iTableExecutor := 0;//IDLE
			
		ELSE
			IF Buffer_Station3.nCount = 0 THEN
				lrTargetLocation := lrStation4Location;
				Buffer_Station4.A_Remove(out => lrStation4Location);
				
			ELSE
				lrTargetLocation := lrStation3Location;
				Buffer_Station3.A_Remove(out => lrStation3Location);
				
			END_IF
			iTableExecutor := 40;
		END_IF
		
	40://
		fbRotaryTable.MR_MoveAbsolute(lrAbsolutePosition := lrTargetLocation);
		IF fbRotaryTable.InPosition THEN
			iTableExecutor := 30;
		END_IF
		
		
END_CASE
///============================================================================================}}}
(* control param *)
fbRobot.ref_CR800.Override:= 5;
uBufferTableCount:= Buffer_RotaryTable.nCount;

(* Mornitoring param *)
bActive 			:= fbRotaryTable.Active;
bBusy				:= fbRotaryTable.Busy;
bError 				:= fbRotaryTable.Error;
iErrorID 			:= fbRotaryTable.ErrorID;
iAxisErrorID 		:= fbRotaryTable.ErrorID;
lrActualPosition 	:= fbRotaryTable.ActualPosition;
rActualVelocity		:= fbRotaryTable.ActualVelocity;
bPowerOn 			:= fbRotaryTable.PowerOn;
bIsHomed 			:= fbRotaryTable.IsHomed;
bInVelocity			:= fbRotaryTable.InVelocity;
bInPostion 			:= fbRotaryTable.InPosition;
bMoveActive 		:= fbRotaryTable.MoveActive;
bJogDone 			:= fbRotaryTable.JogDone;
bStopped 			:= fbRotaryTable.Stopped;
bHalted 			:= fbRotaryTable.Halted;
eStatePlcOpen		:= fbRotaryTable.StatePlcOpen;

fbRobot.ref_CR800.Override:= 30;
fbRotaryTable.Velocity 			:= 50.0;
END_METHOD

METHOD PROTECTED Robot_Process
VAR_INST
	(* Equipment module sequences *)
	RobotState : UINT;
	
END_VAR
CASE RobotState OF	
	0://IDLE go bowl
		fbRobot.MR_GoBowl();
		IF NOT fbRobot.Busy THEN
			RobotState := 5;
		END_IF		
	5://product detected
		IF diProductPresenceBowl.In THEN (* waiting product *)
			RobotState := 6;
		END_IF
	
	6://go input
		fbRobot.MR_GoInputProduct();
		IF NOT fbRobot.Busy THEN
			RobotState := 7;
		END_IF
		
	7://robot pick
		fbRobot.MR_Pick();
		IF NOT fbRobot.Busy THEN
			RobotState := 10;
		END_IF 
		
	10://go to station 1
		fbRobot.MR_GoStation1();
		IF NOT fbRobot.Busy THEN
			RobotState := 20;
		END_IF
		
	20://double trig cam 1+2
		IF doTriggerCam1.Command(PulseWidth:=T#1MS, DelayTimeForSecondTrigger := T#35MS) AND
			doTriggerCam2.Command(PulseWidth:=T#1MS, DelayTimeForSecondTrigger := T#35MS) THEN
			RobotState:= 30;
		END_IF
	30://go to station 2
		fbRobot.MR_GoStation2();
		IF NOT fbRobot.Busy THEN
			RobotState := 40;
		END_IF
	40://double trig cam 3+4
		IF doTriggerCam3.Command(PulseWidth:=T#1MS, DelayTimeForSecondTrigger := T#35MS) AND
			doTriggerCam4.Command(PulseWidth:=T#1MS, DelayTimeForSecondTrigger := T#35MS) THEN
			RobotState := 50;
		END_IF
	50://goto rotary table
		fbRobot.MR_GoRotaryTable();
		IF NOT fbRobot.Busy THEN
			//bProductAboveTable := TRUE;		
			RobotState:= 60;
		END_IF
	60://waiting command from table
		fbRobot.MR_Place();
		IF NOT fbRobot.Busy THEN
			RobotState := 0;
		END_IF
		
END_CASE
END_METHOD

METHOD robotcamtest : BOOL
VAR_INST
	RobotProcess:UINT;
END_VAR
fbRobot.ref_CR800.Override:= 5;
CASE RobotProcess OF
	
	0://IDLE go bowl
		fbRobot.MR_GoBowl();
		IF NOT fbRobot.Busy THEN
			RobotProcess := 5;
		END_IF		
	5://product detected
		IF diProductPresenceBowl.In THEN (* waiting product *)
			RobotProcess := 6;
		END_IF
	
	6://go input
		fbRobot.MR_GoInputProduct();
		IF NOT fbRobot.Busy THEN
			RobotProcess := 7;
		END_IF
		
	7://robot pick
		fbRobot.MR_Pick();
		IF NOT fbRobot.Busy THEN
			RobotProcess := 10;
		END_IF 
		
	10://go to station 1
		fbRobot.MR_GoStation1();
		IF NOT fbRobot.Busy THEN
			RobotProcess := 20;
		END_IF
END_CASE
END_METHOD

PROPERTY Robots : REFERENCE TO FB_Robot
GET
Robots REF= fbRobot;
END_GET
END_PROPERTY

PROPERTY StateInit : REFERENCE TO E_MachineCtrlStateInit
GET
StateInit REF= eMachineStateInit;
END_GET
END_PROPERTY

PROPERTY StateUninitialized : REFERENCE TO E_MachineCtrlStateUninitialized
GET
StateUninitialized REF= eMachineStateUninitialized;
END_GET
END_PROPERTY

METHOD TableProcess : BOOL
VAR_INST
	(*=== Table ===*)
	TableState : UINT;
	OneStep : LREAL:= -61.1928;
	lrRelativeDistance : LREAL;
	
	(* Axis status flags *)
	bActive					: BOOL;
	bBusy					: BOOL;								(* Function block currently executes one of the requests *)
	bError					: BOOL;								(* Error status flag *)
	iErrorID				: UDINT;							(* Error ID *)
	iAxisErrorID			: UDINT;							(* Axis error ID*)
	lrActualPosition		: LREAL;							(* Actual axis position in selected units *)
	rActualVelocity			: REAL;								(* Actual axis velocity in selected units *)
	bPowerOn 				: BOOL;								(* Power On status bit *)
	bIsHomed				: BOOL;								(* Axis has been homed even once *)
	bInVelocity				: BOOL;								(* Axis is moving in target velocity *)
	bInPostion				: BOOL;								(* Axis reached target position *)
	bMoveActive				: BOOL;								(* Axis is moving to target position *)
	bJogDone				: BOOL;								(* Axis manual movement by jog done *)
	bStopped				: BOOL;								(* Axis movement has been stopped *)
	bHalted					: BOOL;								(* Axis movement has been halted *)
	eStatePlcOpen			: E_AxisStatePlcOpen;				(* Current PLCOpen state of axis *)
	
	
	(* Buffer *)
	Buffer_RotaryTable			: FB_DataSetFifo; 	(* Contain the position of all product on the table *)
	Buffer_Station3				: FB_DataSetFifo;	(* Contain the trigger position *)
	Buffer_Station4				: FB_DataSetFifo;	(* Contain the trigger position *)
	
	(*=== Vision ===*)
	Vision3State : UINT;
	Vision4State: UINT;
	lrCapPosStation3 : LREAL;
	lrCapPosStation4: LREAL;
	//lrActualPosition :LREAL;
	bBufferReset : BOOL;
END_VAR
CASE TableState OF
	0://product in
		IF diProductPresenceBowl.In THEN (* waiting product *)
			TableState := 10;
		END_IF
	10://buffer table, station 3, station 4
		IF Buffer_RotaryTable.Add2Data(in1 := OneStep, in2 := OneStep) THEN
			IF Buffer_Station3.Add1Data(in := fbRotaryTable.ActualPosition + OneStep) THEN
				IF Buffer_Station4.Add1Data(in := fbRotaryTable.ActualPosition + 2*OneStep) THEN
					TableState := 20;
		
				END_IF				
			END_IF
		END_IF
	20://take distance
		Buffer_RotaryTable.Remove(out => lrRelativeDistance);
		IF Buffer_RotaryTable.OK THEN
			TableState := 30;
		END_IF
	30://move distance
		fbRotaryTable.MR_MoveRelative(lrRelativeDistance);
		IF fbRotaryTable.InPosition THEN
			TableState := 40;
		END_IF
	40://check
		IF Buffer_RotaryTable.Count >0 THEN
			TableState := 20;
		ELSE 
			TableState := 0;
		END_IF
END_CASE

lrActualPosition := fbRotaryTable.ActualPosition;

CASE Vision3State OF
	0://take capture position
		Buffer_Station3.Remove(out => lrCapPosStation3);
		IF Buffer_Station3.OK THEN
			Vision3State := 10;
		END_IF
	10://waiting table move in pos
		IF LREAL_TO_INT(fbRotaryTable.ActualPosition) = LREAL_TO_INT(lrCapPosStation3) THEN
			Vision3State:= 20;
			
		END_IF
	20://capture
		IF fbRTCVision.M_CommandStation3(PulseWidth:= T#1MS, DelayTimeForSecondTrigger:= T#33MS) THEN
			Vision3State:= 0;
		END_IF

END_CASE

CASE Vision4State OF
	0://take capture position
		Buffer_Station4.Remove(out => lrCapPosStation4);
		IF Buffer_Station4.OK THEN
			Vision4State := 10;
		END_IF
	10://waiting table move in pos
		IF LREAL_TO_INT(fbRotaryTable.ActualPosition) = LREAL_TO_INT(lrCapPosStation4) THEN
			Vision4State:= 20;
			
		END_IF
	20://capture
		IF fbRTCVision.M_CommandStation4(PulseWidth:= T#1MS, DelayTimeForSecondTrigger:= T#33MS) THEN
			Vision4State:= 0;
		END_IF

END_CASE
(*===== Utilities =====*)
IF bBufferReset THEN
	Buffer_Station3.Reset();
	Buffer_Station4.Reset();
	Buffer_RotaryTable.Reset();
//	IF Buffer_Station3.OK AND Buffer_Station4.OK AND Buffer_RotaryTable.OK THEN
		
//	END_IF
END_IF

bActive 			:= fbRotaryTable.Active;
bBusy				:= fbRotaryTable.Busy;
bError 				:= fbRotaryTable.Error;
iErrorID 			:= fbRotaryTable.ErrorID;
iAxisErrorID 		:= fbRotaryTable.ErrorID;
lrActualPosition 	:= fbRotaryTable.ActualPosition;
rActualVelocity		:= fbRotaryTable.ActualVelocity;
bPowerOn 			:= fbRotaryTable.PowerOn;
bIsHomed 			:= fbRotaryTable.IsHomed;
bInVelocity			:= fbRotaryTable.InVelocity;
bInPostion 			:= fbRotaryTable.InPosition;
bMoveActive 		:= fbRotaryTable.MoveActive;
bJogDone 			:= fbRotaryTable.JogDone;
bStopped 			:= fbRotaryTable.Stopped;
bHalted 			:= fbRotaryTable.Halted;
eStatePlcOpen		:= fbRotaryTable.StatePlcOpen;
END_METHOD

METHOD tableRefer : BOOL
VAR_INST
	bparamhome : BOOL;
	bFirstCycle 	: BOOL;
	
	stLiftHomingOptions				: ST_HomingOptions; 

	
	bInit					: BOOL;								(* Power on axis and prepare to work *)
	bAbort					: BOOL;								(* Power off axis and reset status flags *)
	bHome					: BOOL;								(* Home to reference point *)
	bMoveVelocity			: BOOL;								(* Start motion with constant velocity *)
	bMoveAbsolute			: BOOL;								(* Move to absolute position *)
	bMoveAdditive			: BOOL;								(* Move by distance *)
	bMoveRelative			: BOOL;								(* Move by distance *)
	bJog					: BOOL;								(* Start manual jog movement *)
	bStop					: BOOL;								(* High priority stop command *)
	bHalt					: BOOL;								(* Halt current motion, next motion command will abort this command *)
	bReset					: BOOL;								(* Reset axis and return to READY state *)
	
	(* General parameters *)
	bModulo					: BOOL := FALSE;					(* Axis is periodic *)
	lrOverride				: LREAL;							(* Axis velocity override in percents [%] *)
	lrVelocity 				: LREAL;							(* Axis velocirt in measurement units per second *)
	lrAcceleration			: LREAL;							(* Axis acceleration in measurement units per sercond^2 *)
	lrDeceleration 			: LREAL;							(* Axis deceleration in measurement units per sercond^2 *)
	lrJerk					: LREAL;							(* Axis jerk in measurement unit per sercond^3 *)
	lrAbsolutePosition		: LREAL;							(* Target position for MC_MoveAbsolute function *)
	lrRelativeDistance		: LREAL;							(* Relative distance to move for MC_MoveRelative/Additive fuctions *)
	lrHomePosition			: LREAL;							(* This parameters is used to set axis position while performing homing procedure *)
	
	(* Jog function parameters *)	
	lrJogPosition			: LREAL;							(* Relative position to move for jog feature *)
	lrJogVelocity			: LREAL;							(* Jog movement velocity *)
	lrJogAcceleration		: LREAL;							(* Jog movement acceleration *)
	lrJogDeceleration		: LREAL;							(* Jog movement deceleration *)
	lrJogJerk				: LREAL;							(* Jog movement jerk *)
	eJogMode				: E_JogMode;						(* Jog movement mode *)
	eJogDirection			: E_AxisJogDirection;				(* Direction of jog movement *)
	
	(* Stop function parameters *)
	lrStopDeceleration		: LREAL;							(* Stop deceleration *)
	lrStopJerk 				: LREAL;							(* Stop jerk *)
	
	(* Other parameters *)
	stOptions				: ST_MoveOptions;					(* Additional movement options *)
	eDirection				: Tc2_MC2.MC_Direction;				(* Axis movement direction for MC_MoveVelocity *)
	eBufferMode 			: MC_BufferMode := MC_Aborting;		(* Axis buffering mode *)
	
	(* Axis status flags *)
	bActive					: BOOL;
	bBusy					: BOOL;								(* Function block currently executes one of the requests *)
	bError					: BOOL;								(* Error status flag *)
	iErrorID				: UDINT;							(* Error ID *)
	iAxisErrorID			: UDINT;							(* Axis error ID*)
	lrActualPosition		: LREAL;							(* Actual axis position in selected units *)
	rActualVelocity			: REAL;								(* Actual axis velocity in selected units *)
	bPowerOn 				: BOOL;								(* Power On status bit *)
	bIsHomed				: BOOL;								(* Axis has been homed even once *)
	bInVelocity				: BOOL;								(* Axis is moving in target velocity *)
	bInPostion				: BOOL;								(* Axis reached target position *)
	bMoveActive				: BOOL;								(* Axis is moving to target position *)
	bJogDone				: BOOL;								(* Axis manual movement by jog done *)
	bStopped				: BOOL;								(* Axis movement has been stopped *)
	bHalted					: BOOL;								(* Axis movement has been halted *)
	eStatePlcOpen			: E_AxisStatePlcOpen;				(* Current PLCOpen state of axis *)
	
	iAxisStateMachine		: INT;
END_VAR
IF bFirstCycle THEN
	
	lrOverride 			:= 100.0;
	lrVelocity 			:= 100.0;
	lrAcceleration		:= 1500.0;
	lrDeceleration		:= 1500.0;
	lrJerk				:= 1500.0;
	lrAbsolutePosition	:= 0.0;
	lrRelativeDistance	:= 0.0;
	lrHomePosition		:= 0.0;
	
	lrJogPosition		:= 0.0;
	lrJogVelocity 		:= 25.0;
	lrJogAcceleration	:= 250.0;
	lrJogDeceleration	:= 250.0;
	lrJogJerk			:= 250.0;
	
	lrStopDeceleration	:= 250.0;
	lrStopJerk			:= 250.0;	
	
	fbRotaryTable.Override			:= lrOverride;
	fbRotaryTable.Velocity 		:= lrVelocity;
	fbRotaryTable.Acceleration 	:= lrAcceleration;
	fbRotaryTable.Deceleration 	:= lrDeceleration;
	fbRotaryTable.Jerk 			:= lrJerk;
	fbRotaryTable.JogMode			:= eJogMode;
	fbRotaryTable.JogDirection		:= eJogDirection;
	fbRotaryTable.JogVelocity 		:= lrJogVelocity;
	fbRotaryTable.JogAcceleration 	:= lrJogAcceleration;
	fbRotaryTable.JogDeceleration 	:= lrJogDeceleration;
	fbRotaryTable.JogJerk 			:= lrJogJerk;
	fbRotaryTable.StopDeceleration := lrStopDeceleration;
	fbRotaryTable.StopJerk 		:= lrStopJerk;
END_IF

IF bparamhome THEN
	bparamhome := FALSE;
	
	fbRotaryTable.MR_FirstCycle(	sName				:= CONCAT(STR1 := '', STR2 := CONCAT(STR1 := ':', STR2 := '')),
							sMeasurementUnits 	:= '',
							bModulo				:= FALSE);
								
	stLiftHomingOptions.SearchDirection := Tc2_MC2.MC_Direction.MC_Negative_Direction;
	stLiftHomingOptions.SearchVelocity 	:= 50.0;
	stLiftHomingOptions.SyncDirection 	:= Tc2_MC2.MC_Direction.MC_Positive_Direction;
	stLiftHomingOptions.SyncVelocity	:= 10.0;
	
	fbRotaryTable.Override 		:= 100.0;
	fbRotaryTable.Velocity 		:= 50.0;
	fbRotaryTable.Acceleration 	:= 150.0;
	fbRotaryTable.Deceleration 	:= 150.0;
	fbRotaryTable.Jerk 			:= 1500.0;
	fbRotaryTable.HomingMode		:= MC_HomingMode.MC_DefaultHoming;
	fbRotaryTable.HomingOptions 	:= stLiftHomingOptions;
	fbRotaryTable.JogPosition 		:= 0.0;
	fbRotaryTable.JogVelocity 		:= 40.0;
	fbRotaryTable.JogAcceleration 	:= 100.0;
	fbRotaryTable.JogDeceleration 	:= 100.0;
	fbRotaryTable.JogJerk 			:= 1000.0;
	fbRotaryTable.StopDeceleration	:= 100.0;
	fbRotaryTable.StopJerk 		:= 1000.0;

	
END_IF

bActive 			:= fbRotaryTable.Active;
bBusy				:= fbRotaryTable.Busy;
bError 				:= fbRotaryTable.Error;
iErrorID 			:= fbRotaryTable.ErrorID;
iAxisErrorID 		:= fbRotaryTable.ErrorID;
lrActualPosition 	:= fbRotaryTable.ActualPosition;
rActualVelocity		:= fbRotaryTable.ActualVelocity;
bPowerOn 			:= fbRotaryTable.PowerOn;
bIsHomed 			:= fbRotaryTable.IsHomed;
bInVelocity			:= fbRotaryTable.InVelocity;
bInPostion 			:= fbRotaryTable.InPosition;
bMoveActive 		:= fbRotaryTable.MoveActive;
bJogDone 			:= fbRotaryTable.JogDone;
bStopped 			:= fbRotaryTable.Stopped;
bHalted 			:= fbRotaryTable.Halted;
eStatePlcOpen		:= fbRotaryTable.StatePlcOpen;

IF bStop THEN
	bStop := FALSE;
	iAxisStateMachine := 20;
	
ELSIF bHalt THEN
	bHalt := FALSE;
	iAxisStateMachine := 30;
	
ELSIF bReset THEN
	bReset := FALSE;
	iAxisStateMachine := 40;
	
ELSIF bAbort THEN
	bAbort := FALSE;
	iAxisStateMachine := 110;
	
END_IF

CASE iAxisStateMachine OF
	(* Starts seqence *)
	0:
		IF bInit THEN
			bInit := FALSE;
			iAxisStateMachine := 10;

		ELSIF bHome THEN
			bHome := FALSE;
			iAxisStateMachine := 50;
			
		ELSIF bMoveVelocity THEN
			bMoveVelocity := FALSE;
			iAxisStateMachine := 60;
		
		ELSIF bMoveAbsolute THEN
			bMoveAbsolute := FALSE;
			iAxisStateMachine := 70;
		
		ELSIF bMoveAdditive THEN
			bMoveAdditive := FALSE;
			iAxisStateMachine := 80;
			
		ELSIF bMoveRelative THEN
			bMoveRelative := FALSE;
			iAxisStateMachine := 90;
			
		ELSIF bJog THEN
			iAxisStateMachine := 100;
		
		END_IF
		
	(* Initialization *)
	10:
		fbRotaryTable.MR_Init();	
		IF fbRotaryTable.PowerOn THEN
			iAxisStateMachine := 0;
		END_IF
		
	(* Stopping *)
	20:
		bJog := FALSE;
		bMoveAbsolute := FALSE;
		bMoveAdditive := FALSE;
		bMoveRelative := FALSE;
		bMoveVelocity := FALSE;
		
		IF fbRotaryTable.MR_Stop() THEN
			iAxisStateMachine := 0;
		END_IF
		
	(* Halting *)
	30:
		bJog := FALSE;
		bMoveAbsolute := FALSE;
		bMoveAdditive := FALSE;
		bMoveRelative := FALSE;
		bMoveVelocity := FALSE;
		
		fbRotaryTable.MR_Halt();
		IF fbRotaryTable.Halted THEN
			iAxisStateMachine := 0;
		END_IF
		
	(* Resetting *)
	40:
		fbRotaryTable.MR_Reset(); 
		IF NOT fbRotaryTable.Error THEN
			iAxisStateMachine := 0;
		END_IF
	
	(* Homing *)
	50: 
		fbRotaryTable.MR_Home(lrHomePosition:=-2.5);
		IF fbRotaryTable.IsHomed THEN	
			iAxisStateMachine := 0;
		END_IF
	
	(* Move velocity *)	
	60: 
		fbRotaryTable.MR_MoveVelocity();
		IF fbRotaryTable.InVelocity THEN
			iAxisStateMachine := 0;
		END_IF
		
	(* Move absolute *)
	70: 
		fbRotaryTable.MR_MoveAbsolute(lrAbsolutePosition);
		IF fbRotaryTable.InPosition THEN
			iAxisStateMachine := 0;
		END_IF
		
	(* Move additive *)	
	80: 
		fbRotaryTable.MR_MoveAdditive(lrRelativeDistance);
		IF fbRotaryTable.InPosition THEN
			iAxisStateMachine := 0;
		END_IF
		
	(* Move relative *)	
	90: 
		fbRotaryTable.MR_MoveRelative(lrRelativeDistance);
		IF fbRotaryTable.InPosition THEN
			iAxisStateMachine := 0;
		END_IF
		
	(* Jog movement *)	
	100: 
		fbRotaryTable.MR_Jog(bJog);
		IF fbRotaryTable.JogDone THEN
			bJog := FALSE;
			iAxisStateMachine := 0;
		END_IF
		
	(* Deinitialization *)	
	110: 
		fbRotaryTable.MR_Abort();
		IF NOT fbRotaryTable.PowerOn THEN
			iAxisStateMachine := 0;
		END_IF		
END_CASE
END_METHOD

METHOD Test : BOOL
VAR_INST
	(* Robot *)
	RobotState 					: UINT;
	
	(* Table *)
	TableState					: UINT;
	OneStep 					: LREAL:= -60.0; //-61.1928;	(* Define by the distance between station 3 and 4 *)
	lrRelativeDistance 			: LREAL;
	bProductAboveTable 			: BOOL;				(* Signal Robot is at the table *)
	bGetPictureStation3			: BOOL; 			(* Cmd get picture st3 to vision system *)
	bGetPictureStation4 		: BOOL; 			(* Cmd get picture st4 to vision system *)
	bResultProcessing 			: BOOL;				(* Request result from vision system, then add buffer for sorting station *)
	
	(* Buffer *)
	BufferState : UINT;
	Buffer_RotaryTable			: FB_DataSetFifo_1; 	(* Contain the position of all product on the table *)
	Buffer_Station3				: FB_DataSetFifo_1;	(* Contain the trigger position *)
	Buffer_Station4				: FB_DataSetFifo_1;	(* Contain the trigger position *)
	
	(* Sorting Station *)
	Buffer_SortGood				: FB_DataSetFifo_1;
	Buffer_SortDirt				: FB_DataSetFifo_1;
	Buffer_SortDent				: FB_DataSetFifo_1;
	Buffer_SortReject			: FB_DataSetFifo_1;
	
	
	
	lrSortGoodPos				: LREAL;
	lrSortDirtPos				: LREAL;
	lrSortDentPos				: LREAL;
	lrSortRejectPos				: LREAL;
	
	uSortGoodGetPosState		: UINT; 			(* state machine of get sort position from buffer *)
	uSortDirtGetPosState		: UINT;
	uSortDentGetPosState		: UINT;
	uSortRejectGetPosState		: UINT;
		
	tonGoodDelay				: TON;				(* one shoot of good delay valve *)
	tonDirtDelay				: TON;				(* one shoot of dirt delay valve *)
	tonDentDelay				: TON;				(* one shoot of dent delay valve *)								
	tonRejectDelay				: TON;				(* one shoot of reject delay valve *)	
							

	
	(*=== Vision ===*)
	Vision3State 		: UINT;
	Vision4State		: UINT;
	lrCapPosStation3 	: LREAL;
	lrCapPosStation4	: LREAL;
	bGood 				: BOOL;
	bAtVision3 			: BOOL;	(* Product is at vision 3 *)
	bAtVision4 			: BOOL;	(* Product is at vision 4 *)
	eFinalResult		: E_VisionResult;

	(* Axis status flags *)
	bActive					: BOOL;
	bBusy					: BOOL;								(* Function block currently executes one of the requests *)
	bError					: BOOL;								(* Error status flag *)
	iErrorID				: UDINT;							(* Error ID *)
	iAxisErrorID			: UDINT;							(* Axis error ID*)
	lrActualPosition		: LREAL;							(* Actual axis position in selected units *)
	rActualVelocity			: REAL;								(* Actual axis velocity in selected units *)
	bPowerOn 				: BOOL;								(* Power On status bit *)
	bIsHomed				: BOOL;								(* Axis has been homed even once *)
	bInVelocity				: BOOL;								(* Axis is moving in target velocity *)
	bInPostion				: BOOL;								(* Axis reached target position *)
	bMoveActive				: BOOL;								(* Axis is moving to target position *)
	bJogDone				: BOOL;								(* Axis manual movement by jog done *)
	bStopped				: BOOL;								(* Axis movement has been stopped *)
	bHalted					: BOOL;								(* Axis movement has been halted *)
	eStatePlcOpen			: E_AxisStatePlcOpen;
	
	uBufferTableCount : UDINT;
	
	(* testing bit *)
	bResultTest : BOOL;
	bResultGood : BOOL;
	bResultDirt : BOOL;
	bResultDent : BOOL;
	bResultReject : BOOL;

	lrStation3Location : LREAL;
	lrStation4Location : LREAL;
	lrTargetLocation : LREAL;
	
END_VAR
///(*==================================== Robot + Vision process ====================================*){{{
CASE RobotState OF	
	0://IDLE go bowl
		fbRobot.MR_GoBowl();
		IF NOT fbRobot.Busy THEN
			RobotState := 5;
		END_IF		
	5://product detected
		IF diProductPresenceBowl.In THEN (* waiting product *)
			RobotState := 6;
		END_IF
	
	6://go input
		fbRobot.MR_GoInputProduct();
		IF NOT fbRobot.Busy THEN
			RobotState := 7;
		END_IF
		
	7://robot pick
		fbRobot.MR_Pick();
		IF NOT fbRobot.Busy THEN
			RobotState := 10;
		END_IF 
		
	10://go to station 1
		fbRobot.MR_GoStation1();
		IF NOT fbRobot.Busy THEN
			RobotState := 20;
		END_IF
		
	20://double trig cam 1+2
		IF doTriggerCam1.Command(PulseWidth:=T#1MS, DelayTimeForSecondTrigger := T#35MS) AND
			doTriggerCam2.Command(PulseWidth:=T#1MS, DelayTimeForSecondTrigger := T#35MS) THEN
			RobotState:= 30;
		END_IF
	30://go to station 2
		fbRobot.MR_GoStation2();
		IF NOT fbRobot.Busy THEN
			RobotState := 40;
		END_IF
	40://double trig cam 3+4
		IF doTriggerCam3.Command(PulseWidth:=T#1MS, DelayTimeForSecondTrigger := T#35MS) AND
			doTriggerCam4.Command(PulseWidth:=T#1MS, DelayTimeForSecondTrigger := T#35MS) THEN
			RobotState := 50;
		END_IF
	50://goto rotary table
		fbRobot.MR_GoRotaryTable();
		IF NOT fbRobot.Busy THEN
			bProductAboveTable := TRUE;		
			RobotState:= 60;
		END_IF
	60://waiting command from table
		;
		
END_CASE
///============================================================================================}}}
///(*==================================== Table process ====================================*){{{
CASE TableState OF
	0:// idle | waiting for product
		IF bProductAboveTable THEN
			TableState:= 10;
		END_IF
	10://command place product and reset robot sequence
		fbRobot.MR_Place();
		IF NOT fbRobot.Busy THEN
			bProductAboveTable := FALSE;
			RobotState := 0;
			TableState := 20;
		END_IF
	20://add buffer for st 3+4, table
		Buffer_Station3.A_Add(in:= fbRotaryTable.ActualPosition + 2*OneStep); 	(* station position *)
		Buffer_Station4.A_Add(in:= fbRotaryTable.ActualPosition + 4*OneStep);	(* station position *)
		
		Buffer_RotaryTable.A_Add(in:= fbRotaryTable.ActualPosition + OneStep);	(* place position *)
		Buffer_RotaryTable.A_Add(in:= fbRotaryTable.ActualPosition + OneStep);	(* place position *)
		Buffer_RotaryTable.A_Add(in:= fbRotaryTable.ActualPosition + OneStep);	(* place position *)
		Buffer_RotaryTable.A_Add(in:= fbRotaryTable.ActualPosition + OneStep);	(* place position *)
		TableState := 25;
		
	25://CALC POSITION
		IF Buffer_Station3.nCount > 0 AND Buffer_Station4.nCount > 0 THEN
			Buffer_Station3.A_Get(out => lrStation3Location);
			Buffer_Station4.A_Get(out => lrStation4Location);
			
			IF LREAL_TO_LINT(lrStation3Location) > LREAL_TO_LINT(lrStation4Location) THEN
				lrTargetLocation := lrStation3Location;
				Buffer_Station3.A_Remove(out => lrStation3Location);
				
			ELSIF LREAL_TO_LINT(lrStation3Location) < LREAL_TO_LINT(lrStation4Location) THEN
				lrTargetLocation := lrStation4Location;
				Buffer_Station4.A_Remove(out => lrStation4Location);
				
			ELSE
				lrTargetLocation := lrStation3Location;
				Buffer_Station3.A_Remove(out => lrStation3Location);
				Buffer_Station4.A_Remove(out => lrStation4Location);
			
			END_IF
			iTableExecutor := 40;
			
		ELSIF Buffer_Station3.nCount = 0 AND Buffer_Station4.nCount = 0 THEN
			TableState := 0;//IDLE
			
		ELSE
			IF Buffer_Station3.nCount = 0 THEN
				lrTargetLocation := lrStation4Location;
				Buffer_Station4.A_Remove(out => lrStation4Location);
				
			ELSE
				lrTargetLocation := lrStation3Location;
				Buffer_Station3.A_Remove(out => lrStation3Location);
				
			END_IF
			iTableExecutor := 40;
		END_IF
		
//	21://get vision 3capture position
//		IF Vision3State = 0 THEN
//			Vision3State:= 10;
//			TableState:=22;
//		END_IF
//	22://get vision 4 capture position
//		IF Vision4State = 0 THEN
//			Vision4State:= 10;
//			TableState:=30;
//		END_IF
	
	40://MOVE POSITION
		fbRotaryTable.MR_MoveAbsolute(lrAbsolutePosition := lrTargetLocation);
		IF fbRotaryTable.InPosition THEN
			
			TableState := 41;
		END_IF
		
	41:// check position of vision station 3
		IF Vision3State = 0 THEN
			TableState := 42;
		END_IF
	42:
		Buffer_Station3.A_Get(out => lrCapPosStation3);
		bGetPictureStation3 := TRUE;
		
		IF LREAL_TO_INT(fbRotaryTable.ActualPosition) = LREAL_TO_INT(lrCapPosStation3) THEN
			Buffer_Station3.A_Remove(out => lrCapPosStation3);
			Vision3State:= 30;
			TableState := 43;
			
		ELSE
			bGetPictureStation3 := FALSE;
			TableState := 43;
			
		END_IF
			
	43:// check position of vision station 4
		IF Vision4State = 0 THEN
			TableState := 44;
		END_IF
	44:
		Buffer_Station4.A_Get(out => lrCapPosStation4);
		bGetPictureStation4 := TRUE;
		bResultProcessing := TRUE;
		
		IF LREAL_TO_INT(fbRotaryTable.ActualPosition) = LREAL_TO_INT(lrCapPosStation4) THEN
			Buffer_Station4.A_Remove(out => lrCapPosStation4);
			Vision4State:= 30;
			TableState := 60;
			
		ELSE
			bGetPictureStation4 := FALSE;
			bResultProcessing := FALSE;
			TableState := 60;
			
		END_IF
	
	
	
	
//	50://command vision 3
//		IF Vision3State = 0 THEN
//			Vision3State:= 20;
//			TableState:=55;
//		END_IF
//	55:	//command vision 4
//		IF Vision4State = 0 THEN
//			Vision4State:= 20;
//			TableState:=60;
//		END_IF

	
	
	
	
	60://check taking picture done
		IF NOT bGetPictureStation3 AND NOT bGetPictureStation4  AND NOT bResultProcessing THEN
			TableState := 70;
		END_IF
		
	70://state check result | product above table | buffer | go through sorting station
		IF bProductAboveTable THEN
			TableState := 10;//take product
		ELSIF Buffer_RotaryTable.nCount > 0 THEN
			TableState := 30;//get distance
		ELSE
			(* Make sure that the product is sorted *)
			fbRotaryTable.MR_MoveRelative(2*OneStep);
			IF fbRotaryTable.InPosition THEN
				
				TableState := 0;
			END_IF
			
		END_IF
	
END_CASE
///============================================================================================}}}
///(*==================================== Vision 3+4 process ====================================*){{{
CASE Vision3State OF
	0://idle | waiting
		;
//	10://get position in buffer
//		Buffer_Station3.A_Remove(out => lrCapPosStation3);
//		Vision3State := 0;

//	20://check position with table
//		bGetPictureStation3 := TRUE;
//		IF LREAL_TO_INT(fbRotaryTable.ActualPosition) = LREAL_TO_INT(lrCapPosStation3) THEN //convert from lreal to int for less precise
//			Vision3State:= 30;
//		ELSE
//			bGetPictureStation3 := FALSE;
//			Vision3State:= 0;
//		END_IF
			
	30://take picture cam 5+6
		IF doTriggerCam5.Command(PulseWidth:= T#1MS, DelayTimeForSecondTrigger:= T#34MS) AND
			doTriggerCam6.Command(PulseWidth:= T#1MS, DelayTimeForSecondTrigger:= T#34MS) THEN
			
			bGetPictureStation3 := FALSE;
			Vision3State := 0; 
		END_IF
		
END_CASE

(* station 4 have to take picture and request result from system *)
CASE Vision4State OF
	0:
		;
//	10://get trigger position in buffer
//		Buffer_Station4.A_Remove(out => lrCapPosStation4);
//		Vision4State := 0;

//	20://check trigger position with table position
//		bGetPictureStation4 := TRUE;
//		bResultProcessing 	:= TRUE;
//		IF LREAL_TO_INT(fbRotaryTable.ActualPosition) = LREAL_TO_INT(lrCapPosStation4) THEN //convert from lreal to int for less precise
//			Vision4State:= 30;
//		ELSE
//			bResultProcessing			:= FALSE;
//			bGetPictureStation4 		:= FALSE;
//			Vision4State:= 0;
//		END_IF
	
	30://trigger cam 7
		IF doTriggerCam7.Command(PulseWidth:= T#1MS, DelayTimeForSecondTrigger:= T#33MS) THEN
			bGetPictureStation4 := FALSE;
			Vision4State:= 40;
		END_IF
		
	40://request result
		(* testing purpose *)
		bResultGood:= TRUE;
		IF bResultGood THEN
			eFinalResult := VISION_RESULT_GOOD;
			bResultGood := FALSE;
			Vision4State:= 0;
		ELSIF bResultDirt THEN
			eFinalResult := VISION_RESULT_CONTAMINATION_DIRTY;
			bResultDirt := FALSE;
			Vision4State:= 0;
		ELSIF bResultDent THEN
			eFinalResult := VISION_RESULT_SCRATCH_DENT;
			bResultDent := FALSE;
			Vision4State:= 0;
		ELSIF bResultReject THEN
			eFinalResult := VISION_RESULT_REJECT;
			bResultReject := FALSE;
			Vision4State:= 0;
		END_IF

END_CASE
///============================================================================================}}}
///(*==================================== Sorting station ====================================*){{{
(* Add buffer for sorting station *)
CASE eFinalResult OF
	VISION_RESULT_UNKNOWN:
		;
	VISION_RESULT_GOOD:
		Buffer_SortGood.A_Add(in := fbRotaryTable.ActualPosition + lrSortGoodDistance);
		eFinalResult 		:= VISION_RESULT_UNKNOWN;
	VISION_RESULT_CONTAMINATION_DIRTY:
		Buffer_SortDirt.A_Add(in := fbRotaryTable.ActualPosition + lrSortDirtDistance);
		eFinalResult 		:= VISION_RESULT_UNKNOWN;
	VISION_RESULT_SCRATCH_DENT:
		Buffer_SortDent.A_Add(in := fbRotaryTable.ActualPosition + lrSortDentDistance);
		eFinalResult 		:= VISION_RESULT_UNKNOWN;
	VISION_RESULT_REJECT:
		Buffer_SortReject.A_Add(in := fbRotaryTable.ActualPosition + lrSortRejectDistance);
		eFinalResult 		:= VISION_RESULT_UNKNOWN;

END_CASE
(* Shoot the product out *)
(* Good case *)
CASE uSortGoodGetPosState OF
	0://idle | check buffer
		IF Buffer_SortGood.nCount > 0 THEN
			uSortGoodGetPosState:= 10;
		END_IF
	10://get position
		Buffer_SortGood.A_Get(out => lrSortGoodPos);
		uSortGoodGetPosState := 20;
	20://waiting table move in position | command table
		bResultProcessing 	:= FALSE;
		IF LREAL_TO_INT(fbRotaryTable.ActualPosition) <= LREAL_TO_INT(lrSortGoodPos) THEN
			uSortGoodGetPosState := 30;
		END_IF
	30://shoot it
		Buffer_SortGood.A_Remove(out => lrSortGoodPos);
		doBlowGood.Out := TRUE;
		uSortGoodGetPosState := 40;
		
	40://off
		tonGoodDelay(IN := TRUE, PT := tSortValveGoodTime);
		IF tonGoodDelay.Q THEN	
			doBlowGood.Out := FALSE;
			tonGoodDelay.IN := FALSE;
			uSortGoodGetPosState := 0;
		END_IF
		
END_CASE
(* DIRT CASE *)
CASE uSortDirtGetPosState OF
	0://idle | check buffer
		IF Buffer_SortDirt.nCount > 0 THEN
			uSortDirtGetPosState:= 10;
		END_IF
	10://get position
		Buffer_SortDirt.A_Get(out => lrSortDirtPos);
		uSortDirtGetPosState := 20;
	20://waiting table move in position | command table
		bResultProcessing 	:= FALSE;
		IF LREAL_TO_INT(fbRotaryTable.ActualPosition) <= LREAL_TO_INT(lrSortDirtPos) THEN
			uSortDirtGetPosState := 30;
		END_IF
	30://shoot it
		Buffer_SortDirt.A_Remove(out => lrSortDirtPos);
		doBlowDirtScratch.Out := TRUE;
		uSortDirtGetPosState := 40;
		
	40://off
		tonDirtDelay(IN := TRUE, PT := tSortValveDirtTime);
		IF tonDirtDelay.Q THEN	
			doBlowDirtScratch.Out := FALSE;
			tonDirtDelay.IN := FALSE;
			uSortDirtGetPosState := 0;
		END_IF
		
END_CASE
(* DENT CASE *)
CASE uSortDentGetPosState OF
	0://idle | check buffer
		IF Buffer_SortDent.nCount > 0 THEN
			uSortDentGetPosState:= 10;
		END_IF
	10://get position
		Buffer_SortDent.A_Get(out => lrSortDentPos);
		uSortDentGetPosState := 20;
	20://waiting table move in position | command table
		bResultProcessing 	:= FALSE;
		IF LREAL_TO_INT(fbRotaryTable.ActualPosition) <= LREAL_TO_INT(lrSortDentPos) THEN
			uSortDentGetPosState := 30;
		END_IF
	30://shoot it
		Buffer_SortDent.A_Remove(out => lrSortDentPos);
		doBlowDentContamination.Out := TRUE;
		uSortDentGetPosState := 40;
		
	40://off
		tonDentDelay(IN := TRUE, PT := tSortValveDentTime);
		IF tonDentDelay.Q THEN	
			doBlowDentContamination.Out := FALSE;
			tonDentDelay.IN := FALSE;
			uSortDentGetPosState := 0;
		END_IF
		
END_CASE
(* REJECT CASE *)
CASE uSortRejectGetPosState OF
	0://idle | check buffer
		IF Buffer_SortReject.nCount > 0 THEN
			uSortRejectGetPosState:= 10;
		END_IF
	10://get position
		Buffer_SortReject.A_Get(out => lrSortRejectPos);
		uSortRejectGetPosState := 20;
	20://waiting table move in position | command table
		bResultProcessing 	:= FALSE;
		IF LREAL_TO_INT(fbRotaryTable.ActualPosition) <= LREAL_TO_INT(lrSortRejectPos) THEN
			uSortRejectGetPosState := 30;
		END_IF
	30://shoot it
		Buffer_SortReject.A_Remove(out => lrSortRejectPos);
		doBlowReject.Out := TRUE;
		uSortRejectGetPosState := 40;
		
	40://off
		tonRejectDelay(IN := TRUE, PT := tSortValveRejectTime);
		IF tonRejectDelay.Q THEN	
			doBlowReject.Out := FALSE;
			tonRejectDelay.IN := FALSE;
			uSortRejectGetPosState := 0;
		END_IF
		
END_CASE
///============================================================================================}}}
(* control param *)
fbRobot.ref_CR800.Override:= 5;
uBufferTableCount:= Buffer_RotaryTable.nCount;

(* Mornitoring param *)
bActive 			:= fbRotaryTable.Active;
bBusy				:= fbRotaryTable.Busy;
bError 				:= fbRotaryTable.Error;
iErrorID 			:= fbRotaryTable.ErrorID;
iAxisErrorID 		:= fbRotaryTable.ErrorID;
lrActualPosition 	:= fbRotaryTable.ActualPosition;
rActualVelocity		:= fbRotaryTable.ActualVelocity;
bPowerOn 			:= fbRotaryTable.PowerOn;
bIsHomed 			:= fbRotaryTable.IsHomed;
bInVelocity			:= fbRotaryTable.InVelocity;
bInPostion 			:= fbRotaryTable.InPosition;
bMoveActive 		:= fbRotaryTable.MoveActive;
bJogDone 			:= fbRotaryTable.JogDone;
bStopped 			:= fbRotaryTable.Stopped;
bHalted 			:= fbRotaryTable.Halted;
eStatePlcOpen		:= fbRotaryTable.StatePlcOpen;

fbRobot.ref_CR800.Override:= 30;
fbRotaryTable.Velocity 			:= 50.0;
END_METHOD

END_FUNCTION_BLOCK

(* stored: Version 1.1.0.1, ProductVersion 3.1.4024.9
   POU FB_MachineControl: Id {1bd260d7-05fe-41ba-a15a-413659f72f18}, SpecialFunc None
   Folder Internal: Id {8813ce70-337e-4483-a711-2856365d1cdf}
   Folder Properties: Id {29045f01-2b67-43ea-acd9-915a07c376fa}
   Folder References: Id {1ad38fea-3502-4448-beef-6594ebc4effe}
   Folder Status: Id {971e8d7d-8ce9-4462-b8de-cc46e6b1a59b}
   Folder Requests: Id {51769c61-8807-4a83-b47d-198fbacbeb51}
   Folder StateMachine: Id {fcf2a465-15e6-47fd-a8c6-b9a7900c636c}
   Property BowlFeeder: Id {2574449c-1f66-4647-b734-6402fa175952}
   Get Get: Id {389c1fec-9b87-4ee4-9637-69784a171b4f}
   Method GoldenSample: Id {251cea54-20e8-4133-bf48-bd784abd42d0}
   Method M_AutoProcessing: Id {bbfa0667-78a7-4247-a707-1f83fb9a1d16}
   Method MR_Start: Id {443146db-305a-4222-b20b-6401a2c51521}
   Method MR_Stop: Id {45cc0441-f143-4822-b8f2-bcf21d8684b1}
   Method MS_Aborting: Id {7adc3704-59d9-4656-ad31-e25e008f0070}
   Method MS_Auto: Id {9e955c8e-36bd-49e5-a90f-5a0d0edfdf23}
   Method MS_AutoToManual: Id {02d651de-fd64-4bdf-b695-c41b74db33a4}
   Method MS_Emergency: Id {c21af5de-909a-4da8-88d8-257151739074}
   Method MS_Initializing: Id {99a096da-f0d2-4fb3-bcd1-503614bc69d3}
   Method MS_Manual: Id {cfd995b2-d987-47aa-9bb0-1eb8959a8269}
   Method MS_ManualToAuto: Id {bd4c4af3-faf6-45ca-bf78-e8f80721fb97}
   Method MS_ReadyInitialized: Id {b9fb0eda-7ebb-49ea-ace1-57e0fa237813}
   Method MS_Reset: Id {286f95b6-9876-40be-8c77-b17b043cf4d5}
   Method MS_ResetDone: Id {a6caa836-92e0-4931-80a7-2c291a5ebdf0}
   Method MS_Uninitialized: Id {e7564050-17cc-4cfd-9d7a-3500c05b04b7}
   Method Production: Id {57a27725-eff6-400c-8e0e-707934cd22aa}
   Method Production_fixing: Id {4f524830-0d70-4aad-a316-22f5285d8965}
   Method Robot_Process: Id {08e07868-44ca-4ba7-b194-eb2a13c9cadc}
   Method robotcamtest: Id {825274f9-9889-437f-a546-d1f33ad499c6}
   Property Robots: Id {7f945cab-fcf4-42ea-a55f-ae8887eca31e}
   Get Get: Id {da0b5682-da4c-45e1-aecb-4ccc22637b3c}
   Property StateInit: Id {6264ac4e-9149-4997-8345-6779a81ba273}
   Get Get: Id {f3ca5a5b-5318-49aa-b6c3-043b3b74f2e2}
   Property StateUninitialized: Id {ee5f5748-2f92-4c32-baec-09ffa187a7c0}
   Get Get: Id {5f74a4e1-c4bf-4cc8-9020-607d10150e57}
   Method TableProcess: Id {c48c1fc3-cf0e-46c6-86a9-e5a35d25504f}
   Method tableRefer: Id {82184fa1-da82-41ff-b0b5-ab0220bfcbe2}
   Method Test: Id {f5807178-adf8-41e1-a6cd-5cde62a56a97} *)
